// ---- DUTs/ST_DivertConfig.TcDUT
TYPE ST_DivertConfig :
STRUCT
	IntervalToDivert							: UDINT := 1;
	MaxAllowedDivertCount						: UDINT := 4;
	CurrentFunctionCoeffA						: LREAL := 0.5;
	CurrentFunctionCoeffB						: LREAL := 0.17;
	CurrentFunctionCoeffC						: LREAL := 3;
END_STRUCT
END_TYPE;

// ---- DUTs/ST_ExpMoverStatus.TcDUT
TYPE ST_ExpMoverStatus :
STRUCT
	XtsBaseRefData						: REFERENCE TO Tc3_XTS_Utility.ST_PositionInfo;
	HasInterference						: BOOL;
	TrackSectorBndryHeadF			: LREAL;
	TrackSectorBndryTailF			: LREAL;
	TrackSectorCenterHead			: LREAL;
	TrackSectorCenterTail			: LREAL;
	TrackSectorBndryHeadR			: LREAL;
	TrackSectorBndryTailR			: LREAL;
	PartSectorBndryHeadF			: LREAL;
	PartSectorBndryTailF			: LREAL;
	PartSectorCenterHead			: LREAL;
	PartSectorCenterTail			: LREAL;
	PartSectorBndryHeadR			: LREAL;
	PartSectorBndryTailR			: LREAL;
	XtsAdjustedData						: Tc3_XTS_Utility.ST_PositionInfo;
END_STRUCT
END_TYPE

// ---- DUTs/ST_PlcSystem.TcDUT
TYPE ST_PlcSystem :
STRUCT
	nTaskIdx						: DINT;
	nCycleTime					: UDINT;
	TempSysTime					: ULINT;
	SysTime							: ULINT;
	CfgIntervalExec			: UDINT := 2; //x 1 ms task time
END_STRUCT
END_TYPE

// ---- DUTs/ST_SectorsConfig.TcDUT
TYPE ST_SectorsConfig :
STRUCT
	AllSectorsConfig : REFERENCE TO ARRAY[GC.MIN_SECTOR_CT..GC.MAX_SECTOR_CT] OF ST_SectorConfig;
END_STRUCT
END_TYPE

// ---- DUTs/ST_SectorsStatus.TcDUT
TYPE ST_SectorsStatus :
STRUCT
	AllSectorsStatus : REFERENCE TO ARRAY[GC.MIN_SECTOR_CT..GC.MAX_SECTOR_CT] OF ST_SectorStatus;
END_STRUCT
END_TYPE

// ---- DUTs/ST_SwitchStatus.TcDUT
TYPE ST_SwitchStatus :
STRUCT
 	MagnetValue		        AT%Q* 	: INT;
	MagnetEnabled     	        	: BOOL;
    CurrentOutputActual             : LREAL;
    CurrentTheoreticalEstimation    : LREAL;
    CurrentOutputMax                : LREAL;
    PosnCurrentCoeff                : LREAL;
	ShuttleCountAtDivertTrig		: UDINT;
	ShuttleQueueCount				: UDINT;
	ShuttleCountOnShortcut			: UDINT;
END_STRUCT
END_TYPE

// ---- DUTs/ST_SectorConfig.TcDUT
TYPE ST_SectorConfig :
STRUCT
	TrackObjectId			: OTCID;
	PartObjectId	    : OTCID;
	PartObjectIdEnt	    : OTCID;
	PartObjectIdExit    : OTCID;	
	PartSectorStartPosn				: LREAL;
	PartSectorEndPosn				: LREAL;
	TrackSectorStartPosn				: LREAL;
	TrackSectorEndPosn				: LREAL;
	SectorSpansBoundary		: BOOL;
END_STRUCT
END_TYPE

// ---- DUTs/ST_SectorStatus.TcDUT
TYPE ST_SectorStatus :
STRUCT
	MoverIsOnSector			: BOOL;
	MoverCountOnSector		: UDINT;
	MoverEnteredSector		: Tc2_Standard.R_TRIG;
	MoverExitedSector		: Tc2_Standard.F_TRIG;
	SectorLength				: LREAL;
	MoverDistanceFromEnd	: LREAL;
	PercentOfSectorTraversed	: LREAL;
END_STRUCT
END_TYPE

// ---- DUTs/ST_ShortcutConfig.TcDUT
TYPE ST_ShortcutConfig :
STRUCT
	StopAtPowerMat  						: BOOL;
END_STRUCT
END_TYPE

// ---- DUTs/ST_SwitchConfig.TcDUT
TYPE ST_SwitchConfig :
STRUCT
	MagnetOnStartPosition				    : LREAL := 9860; // mm // a little early; 
	MagnetOnEndPosition				    	: LREAL := 10695; // Length of Main Track // mm
	OnInnerLoopOffMagnetPosn				: LREAL	:= 170; //mm
	SwitchCurrentNominal						: LREAL := 5.8; // A (See function for computation)
	CurrentMultFactor							: LREAL := 1310; // Scaling factor for 10V output=25.0A
    UseNominalCurrentVeloSetpoints              : BOOL;
    UseNominalPositionCoeff			            : BOOL := TRUE;
//	PosnCoilResponseTimeCoeffNominal			: LREAL := 0.986;
 	SwitchModeHMI        						: ST_DivertConfig;
 	SwitchModeInternal    						: ST_DivertConfig;
END_STRUCT
END_TYPE;

// ---- DUTs/ST_TrackConfig.TcDUT
TYPE ST_TrackConfig :
STRUCT
	TargetPosnBeforeTrackEnd					: LREAL := 100;
	StopPosPowermat										: LREAL := 7611; // Track Ref; Part Ref ~ 3750 (mm)
	MergeWaitFinishDistance 					: LREAL := 1570;
	MergeWaitAccelDistance						: LREAL; // distance to achieve v_max on the shortcut HD motor region
	ShortcutHDRegionDistance					: LREAL := 2000;
	ShortcutShuttleFullyInPosn 				: LREAL := 1500; // Part Reference (not Track)
	ExpMoverLength										: LREAL := 1200; // roughly 2X SHUTTLE_LENGTH
	MaxLagDistance										: LREAL := 100;
	MergeCollisionRegionDeltaFromL		: LREAL := 2800; // 1715
	MergeCollisionAdvance							: LREAL := 200;
END_STRUCT
END_TYPE

// ---- DUTs/ST_MoverConfig.TcDUT
TYPE ST_MoverConfig EXTENDS ST_MoveOnTrackOptions:
STRUCT
//Velocity (mm/s)
	MaxVelo			: LREAL := 4000;
	NormalVelo		: LREAL := 2700;
	StoppingVelo	: LREAL := 400;
//Acceleration (mm/s^2)
	NormalAccel		: LREAL := MaxVelo;
	MaxAccel		: LREAL := 3*NormalAccel;
//Deceleration (mm/s^2)
	NormalDecel		: LREAL := MaxVelo;	
	MaxDecel		: LREAL := 3*NormalDecel;
//Jerk (mm/s^3)
	NormalJerk		: LREAL := MaxAccel;
	HighJerk			: LREAL := 2*NormalJerk;
	MergeJerk 		: LREAL := 400000;
//Platooning Vars
	VeloComp		: LREAL := 200;
	NormalMoverGap	: LREAL := 750;
	TightMoverGap	: LREAL := 20;
END_STRUCT
END_TYPE

// ---- GVLs/GC.TcGVL
{attribute 'qualified_only'}
VAR_GLOBAL CONSTANT
//Movers-PLC
	nNumMinMovers					: UDINT :=1;
	nNumMaxMovers 					: UDINT :=4; //See General (Persistent, non-constant)

//Movers-MC
	nNumMinMCAxes					: UDINT	:=1;
	nNumMaxMCAxes					: UDINT	:=20;

//Tracks
	nNumMinTracks 					: UDINT :=1; // Do not change - per NC
	OuterFinishPart					: UDINT := 1;
	InnerFinishPart					: UDINT := 2;
	OuterStartPart					: UDINT := 3;	
	nNumMaxTracks 					: UDINT :=3; // Do not change - per NC
	
//Sectors
	MIN_SECTOR_CT										: USINT	:= 1;
	//Make MIN same as first entry
	DIVERTQ_SECTOR_OPART						: USINT := 1;
	DIVERT_DECISION_OPART						: USINT := 2;
	MAG_ON_SECTOR_OPART							: USINT	:= 3; 
	SHORTCUT_ENTRY_SECTOR_IPART 		: USINT := 4; 
	SHORTCUT_ENTRY_HALF_IPART				: USINT := 5; 
	SHORTCUT_CALC_SECTOR_IPART 			: USINT := 6; 
	LOAD_STOP_SECTOR_IPART					: USINT := 7; 
	SHORTCUT_HD_SECTION							: USINT := 8; 
	SHORTCUT_COMPLETE								: USINT := 9; 
	SHORTCUT_EXIT_HALF_IPART				: USINT := 10;
	SHORTCUT_MERGE_COMMAND_WAIT 		: USINT := 11;
	SHORTCUT_MERGE_COMMAND_FLYING 	: USINT := 12;
	SHORTCUT_MERGE_CALC_EXACT 			: USINT := 13;
	INNER_MERGE_TO_FINISH 					: USINT := 14;
	OUTER_SHORTCUT_PROJECTIONFLY		: USINT := 15;
	OUTER_SHORTCUT_PROJECTIONSTAT		: USINT := 16;
	OUTER_PRE_TG_ZONE								: USINT := 17;
	OUTER_TIGHTGAP_ZONE							: USINT := 18;
	OUTER_POST_TG_ZONE							: USINT := 19;
	OUTER_BIGTRACK_END							: USINT := 20;
	OUTER_BIGTRACK_LSMALL						: USINT := 21;
	OUTER_BIGTRACK_MOVE_END					: USINT := 22;
	OUTER_MERGE_COLLISION						: USINT := 23;
	//Make MAX same as last entry
	MAX_SECTOR_CT										: USINT	:= 23;
	
	MIN_TRACKSECTORS_REF : USINT := 1;
	TRACK_SECTORS_STD : USINT := 1;
	TRACK_SECTORS_HEAD : USINT := 2;
	TRACK_SECTORS_TAIL : USINT := 3;
	MAX_TRACKSECTORS_REF : USINT := 3;

	
// Global Position Constants
	SHUTTLE_LENGTH						: LREAL := 600; //mm
END_VAR

// ---- GVLs/GVL_General.TcGVL
VAR_GLOBAL // PERSISTENT
	nNumMovers								: UDINT := 4;
	TotalRuntime							: TIME;
END_VAR

VAR_GLOBAL
	GraphPage												: Tc2_System.T_MaxString := 'https://www.desmos.com/calculator';	

	aStopPositions 									: ARRAY [GC.nNumMinMovers..GC.nNumMaxMovers] OF LREAL;// := [2400, 1700, 1000, 300];

//Configuration
	stMoverConfig										: ST_MoverConfig;
	stTrackGlobalConfig							: ST_TrackConfig;
	stPlanarTrackConfig							: ARRAY[GC.nNumMinTracks..GC.nNumMaxTracks] OF ST_PlanarTrackConfig;
	stTrackShortcutConfig						: ST_ShortcutConfig;
	stSwitchConfig									: ST_SwitchConfig;
	
//XTS - Complete Loop
	XtsCompleteTrackOuterOID				: OTCID := 16#1010480;
	XtsCompleteTrackInnerOID				: OTCID := 16#1010490;
//XTS - Parts
	XtsPartOuterStart								: OTCID := 16#01010020;
	XtsPartInnerFinish							: OTCID := 16#01010170;
	XtsPartOuterFinish							: OTCID := 16#010102C0;
//Planar
	PlanarTrackOuterStart						: OTCID := 16#05120030;
	PlanarTrackInnerFinish					: OTCID := 16#05120020;
	PlanarTrackOuterFinish					: OTCID := 16#05120010;

//Divert
	DivertQueue											: FB_DivertQueue; // Buffer for Divert Requests
	HistoryDivertQueue							: FB_DivertQueue; // Log of all that went through the trigger point
	TempItvlMoverIndex							: UDINT;
	MoverIndexDivertTrig							: UDINT := GC.nNumMinMovers;
	stDivertingMover								: RingBuffer.ST_MoverDivert;
	stMoverDivertInit 							: RingBuffer.ST_MoverDivert; // DO NOT write to this var
	SwitchMagnet										: FB_SwitchMagnet;
	nExitAMoverIsUsingMagnet				: UDINT;
	MagnetControlledByOtherMover		: BOOL;
	ftMagnetControlledByOtherMover	: Tc2_Standard.F_TRIG;
	stSwitchStatus        		    	: ST_SwitchStatus;

//Merge
	MergeQueue											: RingBuffer.RingBufferMoverMerge; // Buffer for Merge events

END_VAR

// ---- GVLs/GVL_Mc3.TcGVL
VAR_GLOBAL	
	TrackSectors					: ARRAY[GC.nNumMinMovers..GC.nNumMaxMovers] OF FB_TrackSectors;
	HeadTrackSectors			: ARRAY[GC.nNumMinMovers..GC.nNumMaxMovers] OF FB_TrackSectors;
	TailTrackSectors			: ARRAY[GC.nNumMinMovers..GC.nNumMaxMovers] OF FB_TrackSectors;
	AllTrackSectors				: FB_AllTrackSectors;

{warning <'bundle FB_Track'>}
	MC_Tracks    		   	 	: ARRAY[GC.nNumMinTracks..GC.nNumMaxTracks] OF Tc3_Mc3PlanarMotion.MC_PlanarTrack;
	MC_Trackfeedback	 		: ARRAY[GC.nNumMinTracks..GC.nNumMaxTracks] OF Tc3_Mc3PlanarMotion.MC_PlanarFeedback;
	TrackTrail 			   		: Tc3_Mc3PlanarMotion.MC_PlanarTrackTrail;
	
{warning <'bundle FB_PlanarMover'>}
	fbPlanarXtsMover			: ARRAY[GC.nNumMinMovers..GC.nNumMaxMovers] OF FB_PlanarXtsMover;
	iMover								: ARRAY[GC.nNumMinMovers..GC.nNumMaxMovers] OF RingBuffer.I_MoverBase;
	aiXpuXtsMover       	: ARRAY[GC.nNumMinMovers..GC.nNumMaxMovers] OF Tc3_XTS_Utility.I_TcIoXtsXpuMover;

	HeadExpMover					: ARRAY[GC.nNumMinMovers..GC.nNumMaxMovers] OF FB_ExpandedMover;
	TailExpMover					: ARRAY[GC.nNumMinMovers..GC.nNumMaxMovers] OF FB_ExpandedMover;
	AllExpMovers					: FB_AllExpMovers;
END_VAR

// ---- ITFs/I_Mover.TcIO
INTERFACE I_Mover (*EXTENDS RingBuffer.I_MoverBase*)

METHOD CycleUpdate : BOOL
VAR_INPUT
END_VAR
END_METHOD

METHOD Init : BOOL
VAR_INPUT
	XtsMover:  I_XtsXlMover1;
	XtsProcessingUnit :  I_XtsProcessingUnit1;
END_VAR
END_METHOD

METHOD JoinNearestTrack : BOOL


VAR

END_VAR
END_METHOD

METHOD LeaveSystemAt : BOOL
VAR_INPUT
	ConnectionOut: REFERENCE TO MC_PlanarTrackConnectionOut;	
END_VAR
END_METHOD

METHOD MoveOnTrack : BOOL
VAR_INPUT
	track: REFERENCE TO MC_PlanarTrack;	
	targetPos: LREAL;
	gap : LREAL; 
	velo : LREAL; 
END_VAR
END_METHOD

PROPERTY MoverOTCID : OTCID
GET
END_GET
SET
END_SET
END_PROPERTY

PROPERTY MoverStopped : BOOL
GET
END_GET
SET
END_SET
END_PROPERTY

PROPERTY P_Dynamics : REFERENCE TO DynamicConstraint_PathXY;
GET
END_GET
END_PROPERTY

PROPERTY P_InSync : Bool
GET
END_GET
END_PROPERTY

PROPERTY P_PlanarFeedback : REFERENCE TO MC_PlanarFeedback
GET
END_GET
END_PROPERTY

PROPERTY P_PlanarMover :   REFERENCE TO  MC_PlanarMover
GET
END_GET
END_PROPERTY

PROPERTY P_TargetTrack : UDINT
GET
END_GET
SET
END_SET
END_PROPERTY

PROPERTY P_TrackSectors : REFERENCE TO FB_TrackSectors
GET
END_GET
SET
END_SET
END_PROPERTY

PROPERTY Rework : BOOL
GET
END_GET
SET
END_SET
END_PROPERTY

METHOD SyncToOtherMover : Bool
VAR_INPUT
	masterSyncPos : LREAL; // Position on the master track
	followerSyncPos : LREAL; // position on the follower track
	PlanarMoverToFollow: REFERENCE TO Tc3_Mc3PlanarMotion.MC_PlanarMover;
	masterTrack : REFERENCE TO Tc3_Mc3PlanarMotion.MC_PlanarTrack; 
	followerTrack : REFERENCE TO Tc3_Mc3PlanarMotion.MC_PlanarTrack; 
	velo : LREAL; 
END_VAR
END_METHOD

METHOD  UpdateXtsTrack
VAR_INPUT
END_VAR
VAR

END_VAR
END_METHOD

PROPERTY XlProcessingUnit : I_XtsProcessingUnit1
GET
END_GET
END_PROPERTY

PROPERTY XtsComFeed : REFERENCE TO  XtsCommandFeedback
GET
END_GET
END_PROPERTY

PROPERTY XtsXlMover :  I_XtsXlMover1
GET
END_GET
END_PROPERTY

END_INTERFACE

// ---- ITFs/I_MoverSector.TcIO
INTERFACE I_MoverSector EXTENDS __SYSTEM.IQueryInterface

PROPERTY P_SectorsConfig : REFERENCE TO ST_SectorsConfig
GET
END_GET
END_PROPERTY

PROPERTY P_SectorsStatus : REFERENCE TO ST_SectorsStatus
GET
END_GET
END_PROPERTY

END_INTERFACE

// ---- POUs/MAIN.TcPOU
PROGRAM MAIN
VAR
	ManMergeCmd				: BOOL;
	bAllDone					: BOOL;
	bStopSequence				: BOOL;
	                    		
	nCase 						: INT;
	nMoveState				  	: ARRAY[GC.nNumMinMovers..GC.nNumMaxMovers] OF INT;
	                    		
	fbXtsEnvironment			: Tc3_XTS_Utility.FB_TcIoXtsEnvironment;
	                    		
	nForCounter					: UDINT;
	M,N,T,Tr					: UDINT;
	dynamics				    : INT;

//Status
	xSimulation					: BOOL := TRUE;
	SystemEnabled				: BOOL;
	stPlcSystem					: ST_PlcSystem;

	IsMoverInBlockingArea		: BOOL;
	nActStopPos					: UINT := 1;
	Fp_error 					: Tc2_Standard.R_TRIG;
	FaultReset					: Tc2_Standard.R_TRIG;
	MoverStop 	AT%I* 			: BOOL;
  ResetSafetyLight AT%Q*      : BOOL;
	MoverStopDone AT%Q*			: BOOL;
	Info 		AT%Q*			: BOOL;
	Operating	AT%Q*			: BOOL;
	Process		AT%Q*			: BOOL;
	Fault		AT%Q*			: BOOL;
	Emergency	AT%Q*			: BOOL;
	                        	
	Voltage1	AT%I*			: UDINT;
	Voltage2	AT%I*			: UDINT;
	                        	
	TcRestart 					: Tc2_Utilities.TC_Restart;
	Restart 					: BOOL;
	busy 						: BOOL;
	fp_start 					: Tc2_Standard.R_TRIG;
	bStartSequence				: BOOL;
	                        	
	Horntimer 					: Tc2_Standard.TP; 
	R_trigHorn 					: Tc2_Standard.R_TRIG;

	StopTime 					: TIME := T#1S;
	StopTimer 					: ARRAY[GC.nNumMinMovers..GC.nNumMaxMovers] OF Tc2_Standard.TON;
	StartTimer 					: ARRAY[GC.nNumMinMovers..GC.nNumMaxMovers] OF BOOL;

	ArcLength 					: ARRAY[GC.nNumMinMovers..GC.nNumMaxMovers] OF LREAL;
	TrackPos					: ARRAY[GC.nNumMinMovers..GC.nNumMaxMovers] OF ARRAY[GC.nNumMinTracks..GC.nNumMaxTracks] OF Tc3_Physics.PositionXYC;
END_VAR

fbXtsEnvironment.Init(bExecute := TRUE);
//Cyclic
M_WritePlanarTrackConfig();
M_UpdateConfigurations();
IF xSimulation THEN
	SystemEnabled	:= TRUE;
ELSE
	SystemEnabled	:= (MoverStop (* SafetyOK *) AND NOT Fault);
END_IF

stPlcSystem.nTaskIdx := GETCURTASKINDEXEX();
IF stPlcSystem.nTaskIdx > 0 THEN
	stPlcSystem.nCycleTime := _TaskInfo[stPlcSystem.nTaskIdx].CycleTime;
	stPlcSystem.SysTime 	:= Tc2_System.F_GetSystemTime();
END_IF

//Command Diverting to Magnet for any designated mover
DivertQueue();
HistoryDivertQueue(); // no removal
MergeQueue();

//Check if any Mover using Magnet;
FOR nExitAMoverIsUsingMagnet :=  GC.nNumMinMovers TO GVL_General.nNumMovers DO
	IF fbPlanarXtsMover[nExitAMoverIsUsingMagnet].P_IsUsingMagnet THEN
		MagnetControlledByOtherMover		:= TRUE;
		EXIT;
	ELSE
		MagnetControlledByOtherMover		:= FALSE;
	END_IF
END_FOR

SwitchMagnet(SafetyPermIntlk := SystemEnabled,
			stSwitchConfig := GVL_General.stSwitchConfig);
ftMagnetControlledByOtherMover(CLK := MagnetControlledByOtherMover);

Emergency :=  MoverStop;
ResetSafetyLight    := NOT MoverStop;

Operating := NOT  MoverStop;
R_trigHorn(clk := Voltage1> 10000 OR Voltage2 >10000);
Horntimer(in:= ( R_trigHorn.Q ) , PT:= T#2S,Q=> info);

IF nCase > 90 THEN
	Process := TRUE;
ELSE 
	Process := FALSE;	
END_IF

IF NOT fbXtsEnvironment.P_IsInitialized THEN
	RETURN;
END_IF

IF NOT MoverStop AND NOT MoverStopDone THEN
	FOR nForCounter:=1 TO nNumMovers DO
		fbPlanarXtsMover[nForCounter].P_Dynamics.SetValuesVADJ(V := stMoverConfig.MaxVelo, A := stMoverConfig.MaxAccel, D := stMoverConfig.MaxDecel, J := stMoverConfig.HighJerk);
		nCase := 140;
		//fbPlanarMover[nForCounter].McPlanarMover.Halt(fbPlanarXtsMover[nForCounter].P_MoverFeedback, fbPlanarXtsMover[nForCounter].P_Dynamics);
	END_FOR		
	MoverStopDone := TRUE;
ELSIF MoverStop THEN
	MoverStopDone := FALSE;
END_IF


TcRestart(
NETID:= '', 
RESTART:= Restart, 
TMOUT:=T#5S , 
BUSY=>busy , 
ERR=> , 
ERRID=> );


fp_start(CLK := bStartSequence);
IF fp_start.Q THEN
	nCase := 10;
	bStartSequence := FALSE;
END_IF

//IsMoverCommandedInShortcut := FALSE;
IsMoverInBlockingArea := FALSE;

bAllDone:= TRUE;
FOR M := GC.nNumMinMovers TO GVL_General.nNumMovers DO///Movers
	StopTimer[M](in:=StartTimer[m],PT:=StopTime);
	GVL_Mc3.fbPlanarXtsMover[M].P_MoverId := M;
	GVL_Mc3.fbPlanarXtsMover[M].P_MoverSort.MoverNumber	:= GVL_Mc3.fbPlanarXtsMover[M].nMoverId;
  GVL_Mc3.aiXpuXtsMover[M]  := fbXtsEnvironment.XpuTcIo(1).MoverTcIo(TO_UINT(M));
  fbPlanarXtsMover[M].iTcIoXtsXpuMover REF= GVL_Mc3.aiXpuXtsMover[M];
	fbPlanarXtsMover[M].Update();
	
	//MoverPos[M].SetValuesXYC(fbPlanarMover[M].McPlanarMover.MCTOPLC.SET.SetPos.x, fbPlanarMover[M].McPlanarMover.MCTOPLC.SET.SetPos.y,fbPlanarMover[M].McPlanarMover.MCTOPLC.SET.SetPos.c);
	
	TR := Tr+1;
	IF Tr = 4 THEN
		Tr :=1;
	END_IF
	{warning <'MoverPhysics does not work'>}
	ArcLength[M] :=GVL_Mc3.MC_Tracks[Tr].GetArcLengthClosestTo(GVL_Mc3.fbPlanarXtsMover[M].P_Physics);
	GVL_Mc3.MC_Tracks[Tr].GetPositionAt(ArcLength[M],TrackPos[M][Tr]);
	
//	IF ABS(GVL_Mc3.fbPlanarXtsMover[M].MoverPhysics.x - TrackPos[M][Tr].x) < 1 AND  ABS(fbPlanarXtsMover[M].MoverPhysics.y - TrackPos[M][Tr].y) < 1 THEN
// 		GVL_Mc3.fbPlanarXtsMover[M].P_XPlanarMover.MoverTrackNr := Tr;
//	END_IF	
	
//	IsMoverCommandedInShortcut := IsMoverCommandedInShortcut OR fbPlanarXtsMover[M].IsCommandedInShortcut;
//	IsMoverInBlockingArea := IsMoverInBlockingArea OR (GVL_Mc3.fbPlanarXtsMover[M].P_PlanarMover.TrackID = GVL_Mc3.MC_Tracks[E_TrackNum.main].MCTOPLC_STD.TrackOID AND 
//														IsBetween(value := GVL_Mc3.fbPlanarXtsMover[M].P_PlanarMover.MoverPos, 
//														minV := GVL_General.stSwitchConfig.fMagnetEntryPosn - GVL_General.stSwitchConfig.MagnetPosnComp, 
//														maxV :=  GVL_General.stSwitchConfig.fMagnetExitPosn + stSwitchConfig.MagnetPosnComp));
	fbPlanarXtsMover[M].P_MoverFeedback.Update();

	Fp_error(CLK := fbPlanarXtsMover[M].P_MC_PlanarMover.Error AND nCase = 100);
	IF Fp_error.Q THEN
		nCase := 140;
		Fault := TRUE;
//		bCmdMagnetOn := FALSE;
	END_IF
END_FOR

FOR T := GC.nNumMinTracks TO GC.nNumMaxTracks DO 
	MC_Tracks[T].Update();
	MC_Trackfeedback[T].Update();
END_FOR

CASE nCase OF
	10:
		Fault := FALSE;
		FOR nForCounter := 1 TO fbXtsEnvironment.XpuTcIo(1).GetPartCount() DO
			fbXtsEnvironment.XpuTcIo(1).PartTcIo(TO_UINT(nForCounter)).TriggerReset();
		END_FOR
		
		nCase := 20;

	20:
		FOR T := GC.nNumMinTracks TO GC.nNumMaxTracks DO 
			MC_Tracks[T].Enable(MC_Trackfeedback[T]);
		END_FOR
				nCase := 30;
		
		
	30: 
		IF MC_Trackfeedback[E_TrackNum.Big].Done AND MC_Trackfeedback[E_TrackNum.Main].Done AND MC_Trackfeedback[E_TrackNum.Small].Done THEN
			nCase := 35;
		END_IF
		
		
	35:
		FOR nForCounter:=GC.nNumMinMovers TO GVL_General.nNumMovers DO
			fbPlanarXtsMover[nForCounter].P_MC_PlanarMover.Reset(fbPlanarXtsMover[nForCounter].P_MoverFeedback);
		END_FOR
		nCase := 36;	
		
		
	36:	
		bAllDone:=TRUE;
		FOR nForCounter:=GC.nNumMinMovers TO GVL_General.nNumMovers DO
			bAllDone:=bAllDone AND fbPlanarXtsMover[nForCounter].P_MoverFeedback.Done;
		END_FOR
		
		IF bAllDone THEN
			nCase := 40;
		END_IF
		
		
	40:
		FOR nForCounter:=GC.nNumMinMovers TO GVL_General.nNumMovers DO
			fbPlanarXtsMover[nForCounter].P_MC_PlanarMover.Enable(fbPlanarXtsMover[nForCounter].P_MoverFeedback);
		END_FOR
		nCase := 50;
	
		
	50:
		bAllDone:=TRUE;
		FOR nForCounter:=GC.nNumMinMovers TO GVL_General.nNumMovers DO
			bAllDone:=bAllDone AND fbPlanarXtsMover[nForCounter].P_MoverFeedback.Done;
		END_FOR
		
		IF bAllDone THEN
			nCase := 60;
		END_IF

	//55:

	60:
		FOR nForCounter:=GC.nNumMinMovers TO GVL_General.nNumMovers DO
			IF nForCounter <= 9 THEN
				fbPlanarXtsMover[nForCounter].JoinTrack(fbPlanarXtsMover[nForCounter].P_MoverFeedback, GVL_Mc3.MC_Tracks[E_TrackNum.Big]);//   Mover[nForCounter].MoverTrackNr]);
			ELSE
				fbPlanarXtsMover[nForCounter].JoinTrack(fbPlanarXtsMover[nForCounter].P_MoverFeedback, GVL_Mc3.MC_Tracks[E_TrackNum.Main]);
			END_IF	
		END_FOR
		
		nCase := 70;
		
	70:
		bAllDone:=TRUE;
		FOR nForCounter:=GC.nNumMinMovers TO GVL_General.nNumMovers DO
			bAllDone:=bAllDone AND fbPlanarXtsMover[nForCounter].P_MoverFeedback.Done;
		END_FOR
		
		IF bAllDone THEN
			nCase := 80;
		END_IF
		
	80:	
		FOR nForCounter:=GC.nNumMinMovers TO GVL_General.nNumMovers DO
			nMoveState[nForCounter] := 0;
			fbPlanarXtsMover[nForCounter].P_MoverOptions.BaseMoveOptions.direction := MC_Direction.mcDirectionPositive;
			fbPlanarXtsMover[nForCounter].P_MoverOptions.BaseMoveOptions.gapMode := MC_GAP_MODE_ON_TRACK.Fast1D;
		END_FOR
		
		nCase := 100;

	100:

		FOR nForCounter:= GC.nNumMinMovers TO GVL_General.nNumMovers DO
			
		//increased accel on shortcut
			IF TrackSectors[nForCounter].SectorStatus[GC.SHORTCUT_HD_SECTION].MoverIsOnSector THEN
				//Increase dynamics on Inner Shortcut
				fbPlanarXtsMover[nForCounter].P_Dynamics.SetValuesVADJ(V := stMoverConfig.NormalVelo, A := stMoverConfig.MaxAccel, D := stMoverConfig.MaxDecel, J := stMoverConfig.HighJerk);
			ELSE
				fbPlanarXtsMover[nForCounter].P_Dynamics.SetValuesVADJ(V := stMoverConfig.NormalVelo, A := stMoverConfig.NormalAccel, D := stMoverConfig.NormalDecel, J := stMoverConfig.NormalJerk);
			END_IF
			

			//Gap Control
			fbPlanarXtsMover[nForCounter].M_EvaluateGap(MoverIndex := nForCounter);

			//Adjust the first mover parameters to induce a platoon
			fbPlanarXtsMover[GC.nNumMinMovers].P_Dynamics.SetValuesVADJ(V := stMoverConfig.NormalVelo-stMoverConfig.VeloComp, A := stMoverConfig.NormalAccel, D := stMoverConfig.NormalDecel, J := stMoverConfig.NormalJerk);

			// allow updating the config per the HMI, when it will not jeopardize the system
			IF NOT TrackSectors[nForCounter].SectorStatus[GC.DIVERT_DECISION_OPART].MoverIsOnSector AND NOT 
				TrackSectors[nForCounter].SectorStatus[GC.SHORTCUT_ENTRY_HALF_IPART].MoverIsOnSector THEN
				stSwitchConfig.SwitchModeInternal		:= 						stSwitchConfig.SwitchModeHMI;
			END_IF
		
			TrackSectors[nForCounter](MoverIndex := nForCounter, MoverRef := iMover[nForCounter]);
//			HeadTrackSectors[nForCounter](MoverIndex := nForCounter, MoverRef := HeadExpMover[nForCounter]);
//			TailTrackSectors[nForCounter](MoverIndex := nForCounter, MoverRef := TailExpMover[nForCounter]);			
			AllTrackSectors(TrackSectorsRef := GVL_Mc3.TrackSectors, HeadTrackSectorsRef := HeadTrackSectors, TailTrackSectorsRef := TailTrackSectors);
			
			HeadExpMover[nForCounter](MoverRef := fbPlanarXtsMover[nForCounter]);
			TailExpMover[nForCounter](MoverRef := fbPlanarXtsMover[nForCounter]);
			AllExpMovers(HeadMoversRef := HeadExpMover, TailMoversRef := TailExpMover);
			
			iMover[nForCounter]	:= fbPlanarXtsMover[nForCounter];
			fbPlanarXtsMover[nForCounter]();
			
			CASE nMoveState[nForCounter] OF
				
				0: // Start-up/Init
					IF fbPlanarXtsMover[nForCounter].P_MoverSort.TrackID = GVL_General.PlanarTrackOuterFinish THEN
						fbPlanarXtsMover[nForCounter].P_MC_PlanarMover.MoveOnTrack(commandFeedback := fbPlanarXtsMover[nForCounter].P_MoverFeedback,
																			targetTrack := GVL_Mc3.MC_Tracks[E_TrackNum.Big],
																			targetPositionOnTrack := GVL_Mc3.MC_Tracks[E_TrackNum.Big].GetLength()-stTrackGlobalConfig.TargetPosnBeforeTrackEnd,
																			constraint := fbPlanarXtsMover[nForCounter].P_Dynamics,
																			options := fbPlanarXtsMover[nForCounter].P_MoverOptions.BaseMoveOptions);
						 nMoveState[nForCounter] 	:= 20;
					ELSIF (fbPlanarXtsMover[nForCounter].P_MoverSort.TrackID = GVL_General.PlanarTrackOuterStart) AND 
								fbPlanarXtsMover[nForCounter].P_XtsPositionInfo.fPartPosition < TrackSectors[nForCounter].P_SectorsConfig[GC.DIVERTQ_SECTOR_OPART].PartSectorStartPosn THEN
						fbPlanarXtsMover[nForCounter].P_MC_PlanarMover.MoveOnTrack(commandFeedback := fbPlanarXtsMover[nForCounter].P_MoverFeedback,
																			targetTrack := GVL_Mc3.MC_Tracks[E_TrackNum.Main],
																			targetPositionOnTrack := GVL_Mc3.MC_Tracks[E_TrackNum.Main].GetLength()-stTrackGlobalConfig.TargetPosnBeforeTrackEnd,
																			constraint := fbPlanarXtsMover[nForCounter].P_Dynamics,
																			options := fbPlanarXtsMover[nForCounter].P_MoverOptions.BaseMoveOptions);
						 nMoveState[nForCounter] 	:= 10;
					END_IF
					
				5: // In Recirc - from Big to Main Track - departing Gap Transition Zone - this Move command could be cyclic
					IF stPlcSystem.TempSysTime = 0 XOR stPlcSystem.TempSysTime = stPlcSystem.SysTime THEN
						stPlcSystem.TempSysTime := stPlcSystem.SysTime + (stPlcSystem.CfgIntervalExec * stPlcSystem.nCycleTime); //next valid clock to issue move command again
						fbPlanarXtsMover[nForCounter].P_eMerge		:= E_MergeType.NoMerge;
						fbPlanarXtsMover[nForCounter].P_MasterSyncId	:= 0;
						fbPlanarXtsMover[nForCounter].P_MasterSyncPosition	:= 0;
						fbPlanarXtsMover[nForCounter].P_MC_PlanarMover.MoveOnTrack(commandFeedback := fbPlanarXtsMover[nForCounter].P_MoverFeedback,
																		targetTrack := GVL_Mc3.MC_Tracks[E_TrackNum.Main],
																		targetPositionOnTrack := GVL_Mc3.MC_Tracks[E_TrackNum.Main].GetLength()-stTrackGlobalConfig.TargetPosnBeforeTrackEnd,
																		constraint := fbPlanarXtsMover[nForCounter].P_Dynamics, 
																		options := fbPlanarXtsMover[nForCounter].P_MoverOptions.BaseMoveOptions);
					END_IF
																		
					//Continuously call the above move command while GapInTransition TRUE (otherwise it's a one-shot command)
					IF NOT fbPlanarXtsMover[nForCounter].P_MoverOptions.GapInTransition THEN
						stPlcSystem.TempSysTime		:= 0;
						nMoveState[nForCounter] 	:= 10;
					END_IF

				10: //Trig state for decision to divert
					IF TrackSectors[nForCounter].afbSector[GC.DIVERTQ_SECTOR_OPART].stSectorStatus.MoverEnteredSector.Q THEN
						GVL_General.stSwitchStatus.ShuttleCountAtDivertTrig		:= GVL_General.stSwitchStatus.ShuttleCountAtDivertTrig +1; //always MODing this; don't need to decrement
						TempItvlMoverIndex	:= ((GVL_General.stSwitchStatus.ShuttleCountAtDivertTrig MOD GVL_General.stSwitchConfig.SwitchModeInternal.IntervalToDivert) +1); // capture the index
					//	AllTrackSectors.M_UpdateSectorCounts(SectorNr := GC.SHORTCUT_CALC_SECTOR_IPART);
						MoverIndexDivertTrig			:= fbPlanarXtsMover[nForCounter].P_MoverId; // regardless of the command to divert, log the MoverID
						DivertQueue.M_UpdateAtTrig();
						nMoveState[nForCounter] 	:= 12;
					END_IF
					
				12: // Command to move needs to be given early
					IF TrackSectors[nForCounter].afbSector[GC.DIVERT_DECISION_OPART].stSectorStatus.MoverEnteredSector.Q THEN
						DivertQueue.RemoveObjFromBuffer();
						nMoveState[nForCounter] 	:= 13;
					END_IF
				
				13:				
				IF (DivertQueue.P_LastObjectRemoved.MoverID <> 0) THEN // Valid MoverID must be obtained by Remove op in previous step
					IF SwitchMagnet.P_PermIntlkOK AND NOT MagnetControlledByOtherMover AND fbPlanarXtsMover[nForCounter].P_CmdDivert AND 
						(fbPlanarXtsMover[nForCounter].P_XtsPositionInfo.fPartPosition < GVL_Mc3.TrackSectors[nForCounter].P_SectorsConfig[GC.MAG_ON_SECTOR_OPART].PartSectorStartPosn)
						AND (stDivertingMover.SysTime <> DivertQueue.P_LastObjectRemoved.SysTime) THEN
							// Divert Move command
							stDivertingMover	:= DivertQueue.P_LastObjectRemoved;
							fbPlanarXtsMover[stDivertingMover.MoverID].P_MC_PlanarMover.MoveOnTrack(commandFeedback := fbPlanarXtsMover[stDivertingMover.MoverID].P_MoverFeedback,
																				targetTrack := GVL_Mc3.MC_Tracks[E_TrackNum.Small],
																				targetPositionOnTrack := (GVL_Mc3.MC_Tracks[E_TrackNum.Small].GetLength() - GC.SHUTTLE_LENGTH) / 2, // midpoint of shortcut
																				constraint := fbPlanarXtsMover[stDivertingMover.MoverID].P_Dynamics,
																				options := fbPlanarXtsMover[stDivertingMover.MoverID].P_MoverOptions.BaseMoveOptions);									
							nMoveState[nForCounter] 	:= 30; //Diverting Mover
					ELSIF NOT fbPlanarXtsMover[nForCounter].P_CmdDivert THEN
							nMoveState[nForCounter] 	:= 15;
					END_IF
				END_IF
	
				15: // In Recirc - from Main to Big Track
					fbPlanarXtsMover[nForCounter].P_MC_PlanarMover.MoveOnTrack(commandFeedback := fbPlanarXtsMover[nForCounter].P_MoverFeedback,
																		targetTrack := GVL_Mc3.MC_Tracks[E_TrackNum.Big],
																		targetPositionOnTrack := GVL_Mc3.MC_Tracks[E_TrackNum.Big].GetLength()-stTrackGlobalConfig.TargetPosnBeforeTrackEnd,
																		constraint := fbPlanarXtsMover[nForCounter].P_Dynamics,
																		options := fbPlanarXtsMover[nForCounter].P_MoverOptions.BaseMoveOptions);
					 nMoveState[nForCounter] 	:= 20;				
					
				20:
					IF TrackSectors[nForCounter].afbSector[GC.OUTER_BIGTRACK_END].stSectorStatus.MoverEnteredSector.Q THEN
						nMoveState[nForCounter]     := 5;
					END_IF				

				30: // Match the move command with the shuttle that is commanded to divert
					SwitchMagnet.M_EvaluateInlineCommands();
					
					IF ftMagnetControlledByOtherMover.Q THEN
						nMoveState[nForCounter] 	:= 40;
					END_IF
			
				40: // Route through shortcut
					IF TrackSectors[nForCounter].afbSector[GC.LOAD_STOP_SECTOR_IPART].stSectorStatus.MoverEnteredSector.Q THEN
						IF stTrackShortcutConfig.StopAtPowerMat THEN
							nMoveState[nForCounter] := 90;
						ELSE
							nMoveState[nForCounter] := 50;
						END_IF					
					END_IF
					
				50: //Pre-Merge state
				IF NOT AllTrackSectors.P_AMoverIsOnSector[GC.OUTER_BIGTRACK_LSMALL] 
						(*AND stSwitchConfig.SwitchModeInternal.MaxAllowedDivertCount = GVL_General.nNumMovers*) THEN
					fbPlanarXtsMover[nForCounter].P_eMerge := E_MergeType.FlyingMergeMoveOnTrack;

					fbPlanarXtsMover[nForCounter].P_MC_PlanarMover.MoveOnTrack(commandFeedback := fbPlanarXtsMover[nForCounter].P_MoverFeedback,
																		targetTrack := GVL_Mc3.MC_Tracks[E_TrackNum.Small],
																		targetPositionOnTrack := GVL_Mc3.MC_Tracks[E_TrackNum.Small].GetLength()-stTrackGlobalConfig.TargetPosnBeforeTrackEnd,
																		constraint := fbPlanarXtsMover[nForCounter].P_Dynamics,
																		options := fbPlanarXtsMover[nForCounter].P_MoverOptions.BaseMoveOptions);

					nMoveState[nForCounter] := 75;
					//Sync to Master ExpMover
				ELSIF TrackSectors[nForCounter].afbSector[GC.SHORTCUT_MERGE_COMMAND_FLYING].stSectorStatus.MoverEnteredSector.Q THEN
					//Nonzero means there is valid Master Mover data
					IF MergeQueue.P_LastObjectRemoved.MoverID <> 0 THEN
					fbPlanarXtsMover[nForCounter].P_eMerge				:= E_MergeType.FlyingMergeMoveSyncd;
						fbPlanarXtsMover[nForCounter].P_MasterSyncId := MergeQueue.P_LastObjectRemoved.MoverID;
//						IF MergeQueue.P_LastObjectRemoved.ExpMoverType = E_ExpMover.Head THEN
//							fbPlanarXtsMover[nForCounter].P_MasterSyncPosition	:= HeadExpMover[fbPlanarXtsMover[nForCounter].P_MasterSyncId].stExpMoverStatus.TrackSectorCenterHead;
//						ELSIF MergeQueue.P_LastObjectRemoved.ExpMoverType = E_ExpMover.Tail THEN
//							fbPlanarXtsMover[nForCounter].P_MasterSyncPosition	:= TailExpMover[fbPlanarXtsMover[nForCounter].P_MasterSyncId].stExpMoverStatus.TrackSectorCenterTail;
//						END_IF
							// use raw mover reference; likely need some position compensation, i.e, stTrackGlobalConfig.ExpMoverLength;
							fbPlanarXtsMover[nForCounter].P_MasterSyncPosition	:= fbPlanarXtsMover[fbPlanarXtsMover[nForCounter].P_MasterSyncId].P_XtsPositionInfo.fTrackPosition;							
						MergeQueue.ClearLastRemoved(); // master sync data consumed by slave
						nMoveState[nForCounter] := 72;					
					END_IF
					
				ELSIF TrackSectors[nForCounter].afbSector[GC.SHORTCUT_MERGE_COMMAND_WAIT].stSectorStatus.MoverEnteredSector.Q OR 
					stTrackShortcutConfig.StopAtPowerMat THEN
					fbPlanarXtsMover[nForCounter].P_eMerge := E_MergeType.MergeFromStaticSyncd;
					
					fbPlanarXtsMover[nForCounter].P_MC_PlanarMover.MoveOnTrack(commandFeedback := fbPlanarXtsMover[nForCounter].P_MoverFeedback,
																		targetTrack := GVL_Mc3.MC_Tracks[E_TrackNum.Small],
																		targetPositionOnTrack := GVL_Mc3.MC_Tracks[E_TrackNum.Small].GetLength()-stTrackGlobalConfig.MergeWaitFinishDistance-stTrackGlobalConfig.MergeWaitAccelDistance,
																		constraint := fbPlanarXtsMover[nForCounter].P_Dynamics,
																		options := fbPlanarXtsMover[nForCounter].P_MoverOptions.BaseMoveOptions);

					nMoveState[nForCounter] := 73;
				END_IF

				60: // Merge - Gear In
 //merge with gap zero
					//issue commmand to sync 
//					masterSyncPos := GVL_Mc.MC_Tracks[E_TrackNum.Big].GetLength()-100;
//					masterPosAtSync := Mover[moverInFront].MoverPos; 
//					followSyncPos := GVL_Mc.MC_Tracks[E_TrackNum.Small].GetLength()-1000;
//					followerPosAtSync :=Mover[1].MoverPos; 
//					fbMover[nForCounter].SyncToOtherMover( 
//						masterSyncPos := masterSyncPos,
//						masterTrack := GVL_Mc.MC_Tracks[E_TrackNum.Big],
//						followerSyncPos := followSyncPos,
//						followerTrack := GVL_Mc.MC_Tracks[e_TrackNum.Small],
//						PlanarMoverToFollow := fbMover[moverInFront].P_PlanarMover,
//						velo:= velo);
//						nMoveState[nForCounter] := 80; 
//					aggressiveDynamics.SetValuesVADJ(4000,4000,8000,400000); 
//					fbMover[nForCounter].P_Dynamics := aggressiveDynamics;
					//fbMover[nForCounter].MoveOnTrack(GVL_Mc.MC_Tracks[E_TrackNum.Main],  GVL_Mc.MC_Tracks[E_TrackNum.Main].GetLength()-500,900,velo);				
				
//					IF fbPlanarXtsMover[nForCounter].P_eMerge <> E_MergeType.NoMerge THEN
						fbPlanarXtsMover[nForCounter].P_Dynamics.SetValuesVADJ(V := stMoverConfig.NormalVelo, A := stMoverConfig.MaxAccel, D := stMoverConfig.MaxDecel, J := stMoverConfig.MergeJerk);
						
						fbPlanarXtsMover[nForCounter].P_MC_PlanarMover.GearInPosOnTrackWithMasterMover(
								commandFeedback:= fbPlanarXtsMover[nForCounter].P_PlanarFeedbackGearMM, 
								masterMover:= fbPlanarXtsMover[fbPlanarXtsMover[nForCounter].P_MasterSyncId].P_MC_PlanarMover,
								trackTrail:= fbPlanarXtsMover[nForCounter].P_SyncTrail,
								masterSyncPosition:= fbPlanarXtsMover[nForCounter].P_MasterSyncPosition,
								masterSyncPositionTrack:= GVL_Mc3.MC_Tracks[E_TrackNum.Big], 
								slaveSyncPosition:= fbPlanarXtsMover[nForCounter].P_XtsPositionInfo.fTrackPosition,
								slaveSyncPositionTrack:= GVL_Mc3.MC_Tracks[E_TrackNum.Small], 
								constraint:= fbPlanarXtsMover[nForCounter].P_Dynamics, 
								options:= fbPlanarXtsMover[nForCounter].P_MoverOptions.GearInMasterMoverOptions);
								nMoveState[nForCounter] := 74;
//					END_IF
						//fbPlanarXtsMover[nForCounter].P_InSync THEN				

				61:
				IF fbPlanarXtsMover[nForCounter].P_MoverFeedback.Done AND ManMergeCmd THEN
					ManMergeCmd	:= FALSE;
					nMoveState[nForCounter] := 75; // 62
				END_IF
					
				62:// Permissive to Merge
//					IF NOT AllTrackSectors.P_AMoverIsOnSector[GC.OUTER_MERGE_COLLISION] THEN
//						nMoveState[nForCounter] := 63;
//					END_IF

				63://Merge from Inner to Outer
//						fbPlanarXtsMover[nForCounter].P_MC_PlanarMover.MoveOnTrack(commandFeedback := fbPlanarXtsMover[nForCounter].P_MoverFeedback,
//																			targetTrack := GVL_Mc3.MC_Tracks[E_TrackNum.Small],
//																			targetPositionOnTrack := GVL_Mc3.MC_Tracks[E_TrackNum.Small].GetLength()-stTrackGlobalConfig.TargetPosnBeforeTrackEnd,
//																			constraint := fbPlanarXtsMover[nForCounter].P_Dynamics,
//																			options := fbPlanarXtsMover[nForCounter].P_MoverOptions.BaseMoveOptions);
//						nMoveState[nForCounter] := 75;
				
				75: //Reset Command On Exit
						IF TrackSectors[nForCounter].afbSector[GC.INNER_MERGE_TO_FINISH].stSectorStatus.MoverEnteredSector.Q THEN
							stSwitchStatus.ShuttleQueueCount := stSwitchStatus.ShuttleQueueCount -1;
							nMoveState[nForCounter] := 5;
						END_IF
				
				90: // Stopped at Powermat Station
					IF fbPlanarXtsMover[nForCounter].P_MoverFeedback.Done THEN
						StartTimer[nForCounter] := TRUE;
						nMoveState[nForCounter] := 100;
					END_IF
					
				100:
					IF StopTimer[nForCounter].Q THEN
						StartTimer[nForCounter] := FALSE;
						nMoveState[nForCounter] := 50;
					END_IF
				END_CASE
		
		END_FOR

		IF bStopSequence AND NOT(IsMoverInBlockingArea) THEN
			nCase := 110;
			bStopSequence := FALSE;
		END_IF
		110:
			N:= nNumMovers;
			FOR nForCounter:=1 TO nNumMovers DO		
				GVL_General.aStopPositions[nForCounter] := TO_LREAL(  fbXtsEnvironment.XpuTcIo(1).MoverTcIo(TO_UINT(N)).GetSimulatedStartUpPosition());
				N := N -1;
			END_FOR
			nCase := 120;
		
		120:	
			nActStopPos := UDINT_TO_UINT(GC.nNumMaxMovers-GVL_General.nNumMovers+1);
			FOR nForCounter:=1 TO nNumMovers DO
				fbPlanarXtsMover[nForCounter].P_Dynamics.SetValuesVADJ(V := stMoverConfig.StoppingVelo, A := stMoverConfig.NormalAccel, D := stMoverConfig.NormalDecel, J := stMoverConfig.NormalJerk);
				nMoveState[nForCounter] := 0;
				fbPlanarXtsMover[nForCounter].P_MC_PlanarMover.MoveOnTrack(fbPlanarXtsMover[nForCounter].P_MoverFeedback, GVL_Mc3.MC_Tracks[E_TrackNum.Main], 300, fbPlanarXtsMover[nForCounter].P_Dynamics, fbPlanarXtsMover[nForCounter].P_MoverOptions.BaseMoveOptions);
			END_FOR

			nCase:= 130; 
		130:
			FOR nForCounter:=1 TO GC.nNumMaxMovers - (GVL_General.nNumMovers-GC.nNumMaxMovers)  DO
				CASE nMoveState[nForCounter] OF
					0:								
						
						IF GVL_Mc3.fbPlanarXtsMover[nForCounter].P_MoverSort.MoverPos < 300 AND GVL_Mc3.fbPlanarXtsMover[nForCounter].P_MoverSort.TrackID = GVL_Mc3.MC_Tracks[E_TrackNum.main].MCTOPLC_STD.TrackOID THEN
							fbPlanarXtsMover[nForCounter].P_MoverOptions.BaseMoveOptions.gap:= stMoverConfig.TightMoverGap;
							fbPlanarXtsMover[nForCounter].P_MC_PlanarMover.MoveOnTrack(commandFeedback := fbPlanarXtsMover[nForCounter].P_MoverFeedback,
																				targetTrack := GVL_Mc3.MC_Tracks[E_TrackNum.Main],
																				targetPositionOnTrack := aStopPositions[nActStopPos],
																				constraint := fbPlanarXtsMover[nForCounter].P_Dynamics,
																				options := fbPlanarXtsMover[nForCounter].P_MoverOptions.BaseMoveOptions);									
							nActStopPos := nActStopPos + 1;
							nMoveState[nForCounter] := 10;
						END_IF
				END_CASE
			END_FOR
		
			bAllDone := TRUE;
			FOR nForCounter:=1 TO nNumMovers DO
				IF NOT(fbPlanarXtsMover[nForCounter].P_MoverFeedback.Done OR fbPlanarXtsMover[nForCounter].P_MoverFeedback.Error) THEN
					bAllDone := FALSE;
					EXIT;
				END_IF
			END_FOR
			
			IF bAllDone THEN
				nCase := 150;
			END_IF
		
		140:
			FOR nForCounter:=1 TO nNumMovers DO
				fbPlanarXtsMover[nForCounter].P_MC_PlanarMover.Halt(fbPlanarXtsMover[nForCounter].P_MoverFeedback, fbPlanarXtsMover[nForCounter].P_Dynamics);
			END_FOR	
			
			nCase := 145;
			
		145:
			bAllDone := TRUE;
			FOR nForCounter:=1 TO nNumMovers DO
				IF NOT(fbPlanarXtsMover[nForCounter].P_MoverFeedback.Done OR fbPlanarXtsMover[nForCounter].P_MoverFeedback.Error) THEN
					bAllDone := FALSE;
					EXIT;
				END_IF
			END_FOR
			
			IF bAllDone THEN
				nCase := 150;
			END_IF
		
		//Disable
		150:
			FOR nForCounter:=1 TO nNumMovers DO
				fbPlanarXtsMover[nForCounter].P_MC_PlanarMover.Disable(fbPlanarXtsMover[nForCounter].P_MoverFeedback);
			END_FOR
				
			nCase := 0;
END_CASE

FaultReset(CLK := MoverStop);

IF FaultReset.Q THEN
	Fault	:= FALSE;
END_IF

METHOD M_UpdateConfigurations
stTrackGlobalConfig.MergeWaitAccelDistance := 
F_PosnDisp(Accel := stMoverConfig.MaxAccel, 
								VeloFinal := stMoverConfig.NormalVelo, 
								VeloInit := 0);
END_METHOD

METHOD M_WritePlanarTrackConfig
stPlanarTrackConfig[E_TrackNum.Big].MCTrack				:= GVL_Mc3.MC_Tracks[E_TrackNum.Big].MCTOPLC_STD;
stPlanarTrackConfig[E_TrackNum.Small].MCTrack			:= GVL_Mc3.MC_Tracks[E_TrackNum.Small].MCTOPLC_STD;
stPlanarTrackConfig[E_TrackNum.Main].MCTrack			:= GVL_Mc3.MC_Tracks[E_TrackNum.Main].MCTOPLC_STD;
                                                    	
stPlanarTrackConfig[E_TrackNum.Big].TrackIndex			:= E_TrackNum.Big;
stPlanarTrackConfig[E_TrackNum.Small].TrackIndex		:= E_TrackNum.Small;
stPlanarTrackConfig[E_TrackNum.Main].TrackIndex			:= E_TrackNum.Main;
END_METHOD

END_PROGRAM

// ---- POUs/FUNs/F_PosnDisp.TcPOU
FUNCTION F_PosnDisp : LREAL
VAR_INPUT
	VeloInit 	: LREAL;
	VeloFinal	: LREAL;
	Accel		: LREAL;
END_VAR
VAR
END_VAR

IF Accel <> 0 THEN
	F_PosnDisp := (EXPT(VeloFinal,2) - EXPT(VeloInit,2)) / (2*Accel);
END_IF

END_FUNCTION

// ---- POUs/FBs/FB_DivertQueue.TcPOU
FUNCTION_BLOCK FB_DivertQueue EXTENDS RingBuffer.RingBufferMoverDivert
VAR
//	nForCounterInterval			: UDINT;
	MoverDivert							: RingBuffer.ST_MoverDivert;
END_VAR

METHOD M_UpdateAtTrig
VAR_INST
	stDivertLogMover								: RingBuffer.ST_MoverDivert;
END_VAR
stDivertLogMover.MoverID							:= MoverIndexDivertTrig;
IF (stSwitchStatus.ShuttleQueueCount < GVL_General.stSwitchConfig.SwitchModeInternal.MaxAllowedDivertCount) THEN // permissives to allow a mover to divert
		stDivertLogMover.Divert								:= RingBuffer.E_Divert.Divert;
	IF (TempItvlMoverIndex = GVL_General.stSwitchConfig.SwitchModeInternal.IntervalToDivert) THEN
		stDivertLogMover.DivertOnInterval													:= TRUE;
		stSwitchStatus.ShuttleQueueCount := stSwitchStatus.ShuttleQueueCount + 1;
		fbPlanarXtsMover[stDivertLogMover.MoverID].P_CmdDivert		:= (stDivertLogMover.Divert = RingBuffer.E_Divert.Divert) AND stDivertLogMover.DivertOnInterval;
		HistoryDivertQueue.AddObjToBuffer(RefObject := stDivertLogMover);
	END_IF
END_IF

DivertQueue.AddObjToBuffer(RefObject := stDivertLogMover);
stDivertLogMover					:= stMoverDivertInit;
END_METHOD

PROPERTY P_MoverDivert : REFERENCE TO ST_MoverDivert
GET
P_MoverDivert REF= MoverDivert;
END_GET
END_PROPERTY

END_FUNCTION_BLOCK

// ---- POUs/FBs/FB_SwitchMagnet.TcPOU
FUNCTION_BLOCK FB_SwitchMagnet

VAR_INPUT
	stSwitchConfig				: REFERENCE TO ST_SwitchConfig := GVL_General.stSwitchConfig;
	ShuttleVelocity				: REFERENCE TO LREAL := GVL_General.stMoverConfig.NormalVelo;
	SafetyPermIntlk				: REFERENCE TO BOOL;
END_VAR
//VAR_IN_OUT
//	MoverRef						: 
//END_VAR
VAR
	TimeoutTime					: TIME := T#3S;
	pwm							: FB_PWM;
	Command	 		  			: BOOL;
	Timeout						: TON;
	PermIntlkOK					: BOOL;
END_VAR
VAR_OUTPUT
	MagnetIsOn					: BOOL;
END_VAR

_M_EvaluatePermIntlk();
_M_EvaluateCommands();

//Configuration
IF GVL_General.stSwitchConfig.UseNominalCurrentVeloSetpoints THEN
    GVL_General.stSwitchStatus.CurrentTheoreticalEstimation     := GVL_General.stSwitchConfig.SwitchCurrentNominal;
ELSE
    GVL_General.stSwitchStatus.CurrentTheoreticalEstimation     := F_CurrentVelocity(Velocity := GVL_General.stMoverConfig.NormalVelo, a := GVL_General.stSwitchConfig.SwitchModeHMI.CurrentFunctionCoeffA, b := GVL_General.stSwitchConfig.SwitchModeHMI.CurrentFunctionCoeffB, c := GVL_General.stSwitchConfig.SwitchModeHMI.CurrentFunctionCoeffC);
END_IF

GVL_General.stSwitchStatus.CurrentOutputMax     := GVL_General.stSwitchStatus.CurrentTheoreticalEstimation;

//Output
IF PermIntlkOK AND Command THEN
	GVL_General.stSwitchStatus.MagnetValue := LREAL_TO_INT(GVL_General.stSwitchStatus.CurrentOutputMax*stSwitchConfig.CurrentMultFactor);
ELSE
	GVL_General.stSwitchStatus.MagnetValue := 0;
END_IF

MagnetIsOn	:= (GVL_General.stSwitchStatus.MagnetValue > 0);

IF stSwitchConfig.CurrentMultFactor <> 0 THEN
    GVL_General.stSwitchStatus.CurrentOutputActual  := GVL_General.stSwitchStatus.MagnetValue / stSwitchConfig.CurrentMultFactor;
END_IF

pwm();

//Use Magnet feedback to this timer; set preset time based on mover velocity
Timeout(IN := MagnetIsOn, PT := TimeoutTime);

METHOD PRIVATE _M_EvaluateCommands
VAR_INST
	nForCounter		: UDINT;
END_VAR
IF NOT PermIntlkOK OR Timeout.Q THEN
	Command		:= FALSE;
END_IF
END_METHOD

METHOD PRIVATE _M_EvaluatePermIntlk
PermIntlkOK	:= SafetyPermIntlk AND NOT Timeout.Q;
END_METHOD

METHOD M_EvaluateInlineCommands
IF stDivertingMover.MoverID <> 0 THEN
	IF GVL_Mc3.TrackSectors[stDivertingMover.MoverID].SectorStatus[GC.MAG_ON_SECTOR_OPART].MoverIsOnSector THEN
		Command								:= TRUE;
		fbPlanarXtsMover[stDivertingMover.MoverID].P_IsUsingMagnet := TRUE;
	ELSIF GVL_Mc3.TrackSectors[stDivertingMover.MoverID].SectorStatus[GC.MAG_ON_SECTOR_OPART].MoverExitedSector.Q THEN
		Command								:= FALSE; // Any mover exiting the Magnet drops the command
		fbPlanarXtsMover[stDivertingMover.MoverID].P_CmdDivert			:= FALSE;
		fbPlanarXtsMover[stDivertingMover.MoverID].P_IsUsingMagnet 	:= FALSE;
	END_IF
END_IF
END_METHOD

PROPERTY P_PermIntlkOK : BOOL
GET
P_PermIntlkOK := PermIntlkOK;
END_GET
SET
PermIntlkOK := P_PermIntlkOK;
END_SET
END_PROPERTY

END_FUNCTION_BLOCK

// ---- POUs/FUNs/F_CurrentVelocity.TcPOU
FUNCTION F_CurrentVelocity : LREAL
VAR_INPUT
    Velocity    : LREAL;
	a			: LREAL := 1.1;
	b			: LREAL := 0.1;
	c			: LREAL := 5.8;
END_VAR

F_CurrentVelocity  := a*EXPT((Velocity/1000),2) + b*(Velocity/1000) + c;

END_FUNCTION

// ---- POUs/FBs/FB_TrackSectors.TcPOU
FUNCTION_BLOCK FB_TrackSectors IMPLEMENTS I_MoverSector
// VAR_INPUT
// END_VAR                
VAR                    
//	InitDone						: BOOL;
	SectorIndex						: UDINT;
                       
//Configurations       
	SectorConfig					: ARRAY[GC.MIN_SECTOR_CT..GC.MAX_SECTOR_CT] OF ST_SectorConfig;
	SectorsConfig					: ST_SectorsConfig;
                       
	afbSector								: ARRAY[GC.MIN_SECTOR_CT..GC.MAX_SECTOR_CT] OF FB_TrackSector;
	
	LinkedMoveList 				: ARRAY[GC.MIN_SECTOR_CT..GC.MAX_SECTOR_CT] OF RingBuffer.RingBufferLinkedListEntry;
	iMover								: RingBuffer.ST_IDLinkedListEntry;
END_VAR
VAR_IN_OUT
	MoverIndex						: UDINT;
	MoverRef						: RingBuffer.I_MoverBase; // I_Mover
END_VAR
VAR_OUTPUT
	SectorStatus					: ARRAY[GC.MIN_SECTOR_CT..GC.MAX_SECTOR_CT] OF ST_SectorStatus;
	SectorsStatus					: ST_SectorsStatus;
END_VAR

//IF NOT InitDone THEN
	_M_Configurations();
//END_IF

iMover.iMover := MoverRef;

_M_UpdateStatus();

FOR SectorIndex := GC.MIN_SECTOR_CT TO GC.MAX_SECTOR_CT DO
	//SectorLists
	LinkedMoveList[SectorIndex]();	

	//Planar Mover
	afbSector[SectorIndex].P_MoverSort			:= GVL_Mc3.fbPlanarXtsMover[MoverIndex].P_MoverSort;

	//XTS Mover Reference
	IF MoverRef <> 0 THEN
		afbSector[SectorIndex].P_XtsPositionInfo		:= MoverRef.P_XtsPositionInfo;
	END_IF
	
	//Sector Configuration
	afbSector[SectorIndex].P_TrackSectorConfig	:= SectorConfig[SectorIndex];

	//FB calls
	afbSector[SectorIndex](refPlanarTracks := GVL_General.stPlanarTrackConfig);
END_FOR

METHOD _M_Configurations
IF (GVL_General.XtsCompleteTrackOuterOID <> 0) AND (GVL_General.XtsCompleteTrackInnerOID <> 0) THEN

{warning <'Make this a function of velocity; it's not that sensitive to current'>}
//IF GVL_General.stSwitchConfig.UseNominalPositionCoeff THEN
//	GVL_General.stSwitchStatus.PosnCurrentCoeff                                 := GVL_General.stSwitchConfig.PosnCoilResponseTimeCoeffNominal;
//ELSE (* NOT GVL_General.stSwitchConfig.UseHMINominalSetpoints *)
//	GVL_General.stSwitchStatus.PosnCurrentCoeff                                 := PositionF_CurrentCoeff(Current := GVL_General.stSwitchStatus.CurrentOutputMax);
//END_IF

	SectorConfig[GC.DIVERTQ_SECTOR_OPART].PartObjectId								:= GVL_General.XtsPartOuterStart;
	SectorConfig[GC.DIVERTQ_SECTOR_OPART].PartSectorStartPosn				:= SectorConfig[GC.DIVERT_DECISION_OPART].PartSectorStartPosn - GC.SHUTTLE_LENGTH;
	SectorConfig[GC.DIVERTQ_SECTOR_OPART].PartSectorEndPosn			 		:= SectorConfig[GC.DIVERT_DECISION_OPART].PartSectorStartPosn;
	SectorConfig[GC.DIVERTQ_SECTOR_OPART].TrackSectorStartPosn				:= 0; 
	SectorConfig[GC.DIVERTQ_SECTOR_OPART].TrackSectorEndPosn 				:= 0;

	SectorConfig[GC.DIVERT_DECISION_OPART].PartObjectId						:= GVL_General.XtsPartOuterStart;
	SectorConfig[GC.DIVERT_DECISION_OPART].PartSectorStartPosn			:= F_PosnInitial(VeloInit := GVL_General.stMoverConfig.NormalVelo, VeloFinal := 0, Accel := GVL_General.stMoverConfig.NormalDecel, PosnFinal := SectorConfig[GC.MAG_ON_SECTOR_OPART].PartSectorStartPosn);
	SectorConfig[GC.DIVERT_DECISION_OPART].PartSectorEndPosn			 	:= SectorConfig[GC.MAG_ON_SECTOR_OPART].PartSectorStartPosn;
	SectorConfig[GC.DIVERT_DECISION_OPART].TrackSectorStartPosn			:= 0; 
	SectorConfig[GC.DIVERT_DECISION_OPART].TrackSectorEndPosn 			:= 0;

	SectorConfig[GC.MAG_ON_SECTOR_OPART].PartObjectId						:= GVL_General.XtsPartOuterStart;
	SectorConfig[GC.MAG_ON_SECTOR_OPART].PartSectorStartPosn			:= GVL_General.stSwitchConfig.MagnetOnStartPosition;
	SectorConfig[GC.MAG_ON_SECTOR_OPART].PartSectorEndPosn			 	:= GVL_General.stSwitchConfig.MagnetOnEndPosition;
	SectorConfig[GC.MAG_ON_SECTOR_OPART].TrackSectorStartPosn			:= GVL_General.stSwitchConfig.MagnetOnStartPosition;
	SectorConfig[GC.MAG_ON_SECTOR_OPART].TrackSectorEndPosn 			:= GVL_General.stSwitchConfig.MagnetOnEndPosition;
	SectorConfig[GC.MAG_ON_SECTOR_OPART].SectorSpansBoundary			:= FALSE; 	
	
	SectorConfig[GC.SHORTCUT_ENTRY_SECTOR_IPART].PartObjectId					:= GVL_General.XtsPartInnerFinish;
	SectorConfig[GC.SHORTCUT_ENTRY_SECTOR_IPART].PartSectorStartPosn			:= 0;
	SectorConfig[GC.SHORTCUT_ENTRY_SECTOR_IPART].PartSectorEndPosn			:= stTrackGlobalConfig.ShortcutShuttleFullyInPosn;
	SectorConfig[GC.SHORTCUT_ENTRY_SECTOR_IPART].TrackSectorStartPosn		:= 0;
	SectorConfig[GC.SHORTCUT_ENTRY_SECTOR_IPART].TrackSectorEndPosn 			:= 0;

	SectorConfig[GC.SHORTCUT_ENTRY_HALF_IPART].PartObjectId						:= GVL_General.XtsPartInnerFinish;
	SectorConfig[GC.SHORTCUT_ENTRY_HALF_IPART].PartSectorStartPosn			:= 0;
	SectorConfig[GC.SHORTCUT_ENTRY_HALF_IPART].PartSectorEndPosn			 	:= (GVL_Mc3.MC_Tracks[E_TrackNum.Small].GetLength() / 2);
	SectorConfig[GC.SHORTCUT_ENTRY_HALF_IPART].TrackSectorStartPosn			:= 0;
	SectorConfig[GC.SHORTCUT_ENTRY_HALF_IPART].TrackSectorEndPosn 			:= 0;

	SectorConfig[GC.SHORTCUT_CALC_SECTOR_IPART].PartObjectId						:= GVL_General.XtsPartInnerFinish;
	SectorConfig[GC.SHORTCUT_CALC_SECTOR_IPART].PartSectorStartPosn			:= 0;
	SectorConfig[GC.SHORTCUT_CALC_SECTOR_IPART].PartSectorEndPosn			:= GVL_Mc3.MC_Tracks[E_TrackNum.Small].GetLength()-stTrackGlobalConfig.MergeWaitFinishDistance + (stMoverConfig.NormalMoverGap /2);
	SectorConfig[GC.SHORTCUT_CALC_SECTOR_IPART].TrackSectorStartPosn			:= 0;
	SectorConfig[GC.SHORTCUT_CALC_SECTOR_IPART].TrackSectorEndPosn 			:= 0;

	SectorConfig[GC.LOAD_STOP_SECTOR_IPART].PartObjectId						    := GVL_General.XtsPartInnerFinish;
	SectorConfig[GC.LOAD_STOP_SECTOR_IPART].PartSectorStartPosn			    := F_PosnInitial(VeloInit := GVL_General.stMoverConfig.NormalVelo, VeloFinal := 0, Accel := GVL_General.stMoverConfig.NormalDecel, PosnFinal := (GVL_Mc3.MC_Tracks[E_TrackNum.Small].GetLength() /2) -GC.SHUTTLE_LENGTH);
	SectorConfig[GC.LOAD_STOP_SECTOR_IPART].PartSectorEndPosn			 	:= GC.SHUTTLE_LENGTH + (GVL_Mc3.MC_Tracks[E_TrackNum.Small].GetLength() /2) ;
	SectorConfig[GC.LOAD_STOP_SECTOR_IPART].TrackSectorStartPosn			    := 0;
	SectorConfig[GC.LOAD_STOP_SECTOR_IPART].TrackSectorEndPosn 			 	:= 0;

	SectorConfig[GC.SHORTCUT_COMPLETE].PartObjectId													:= GVL_General.XtsPartInnerFinish;
	SectorConfig[GC.SHORTCUT_COMPLETE].PartSectorStartPosn								:= 0;
	SectorConfig[GC.SHORTCUT_COMPLETE].PartSectorEndPosn								:= GVL_Mc3.MC_Tracks[E_TrackNum.Small].GetLength();
	SectorConfig[GC.SHORTCUT_COMPLETE].TrackSectorStartPosn						:= 0;
	SectorConfig[GC.SHORTCUT_COMPLETE].TrackSectorEndPosn 							:= 0;
	
	SectorConfig[GC.SHORTCUT_HD_SECTION].PartObjectId										:= GVL_General.XtsPartInnerFinish;
	SectorConfig[GC.SHORTCUT_HD_SECTION].PartSectorStartPosn							:= stTrackGlobalConfig.ShortcutHDRegionDistance;
	SectorConfig[GC.SHORTCUT_HD_SECTION].PartSectorEndPosn								:= GVL_Mc3.MC_Tracks[E_TrackNum.Small].GetLength()-stTrackGlobalConfig.ShortcutHDRegionDistance;
	SectorConfig[GC.SHORTCUT_HD_SECTION].TrackSectorStartPosn						:= 0;
	SectorConfig[GC.SHORTCUT_HD_SECTION].TrackSectorEndPosn 							:= 0;
	
	SectorConfig[GC.SHORTCUT_EXIT_HALF_IPART].PartObjectId										:= GVL_General.XtsPartInnerFinish;
	SectorConfig[GC.SHORTCUT_EXIT_HALF_IPART].PartSectorStartPosn				:= (GVL_Mc3.MC_Tracks[E_TrackNum.Small].GetLength() / 2);
	SectorConfig[GC.SHORTCUT_EXIT_HALF_IPART].PartSectorEndPosn			 		:= GVL_Mc3.MC_Tracks[E_TrackNum.Small].GetLength();
	SectorConfig[GC.SHORTCUT_EXIT_HALF_IPART].TrackSectorStartPosn				:= 0;
	SectorConfig[GC.SHORTCUT_EXIT_HALF_IPART].TrackSectorEndPosn 				:= 0;

	SectorConfig[GC.SHORTCUT_MERGE_COMMAND_WAIT].PartObjectId								:= GVL_General.XtsPartInnerFinish;
	SectorConfig[GC.SHORTCUT_MERGE_COMMAND_WAIT].PartSectorStartPosn					:= F_PosnInitial(VeloInit := GVL_General.stMoverConfig.NormalVelo, VeloFinal := 0, Accel := GVL_General.stMoverConfig.NormalDecel, PosnFinal := (GVL_Mc3.MC_Tracks[E_TrackNum.Small].GetLength()-stTrackGlobalConfig.MergeWaitFinishDistance-stTrackGlobalConfig.MergeWaitAccelDistance));
	SectorConfig[GC.SHORTCUT_MERGE_COMMAND_WAIT].PartSectorEndPosn						:= GVL_Mc3.MC_Tracks[E_TrackNum.Small].GetLength()-stTrackGlobalConfig.MergeWaitFinishDistance + (GC.SHUTTLE_LENGTH /2);
	SectorConfig[GC.SHORTCUT_MERGE_COMMAND_WAIT].TrackSectorStartPosn					:= 0;
	SectorConfig[GC.SHORTCUT_MERGE_COMMAND_WAIT].TrackSectorEndPosn 					:= 0;
	
	SectorConfig[GC.SHORTCUT_MERGE_COMMAND_FLYING].PartObjectId								:= GVL_General.XtsPartInnerFinish;
	SectorConfig[GC.SHORTCUT_MERGE_COMMAND_FLYING].PartSectorStartPosn					:= SectorConfig[GC.SHORTCUT_MERGE_COMMAND_WAIT].PartSectorStartPosn - GC.SHUTTLE_LENGTH;
	SectorConfig[GC.SHORTCUT_MERGE_COMMAND_FLYING].PartSectorEndPosn						:= SectorConfig[GC.SHORTCUT_MERGE_COMMAND_WAIT].PartSectorStartPosn;
	SectorConfig[GC.SHORTCUT_MERGE_COMMAND_FLYING].TrackSectorStartPosn				:= 0;
	SectorConfig[GC.SHORTCUT_MERGE_COMMAND_FLYING].TrackSectorEndPosn 					:= 0;

	//for calculation of length in the "3rd condition"
	SectorConfig[GC.SHORTCUT_MERGE_CALC_EXACT].PartObjectId										:= GVL_General.XtsPartInnerFinish;
	SectorConfig[GC.SHORTCUT_MERGE_CALC_EXACT].PartSectorStartPosn					:= F_PosnInitial(VeloInit := GVL_General.stMoverConfig.NormalVelo, VeloFinal := 0, Accel := GVL_General.stMoverConfig.NormalDecel, PosnFinal := (GVL_Mc3.MC_Tracks[E_TrackNum.Small].GetLength()-stTrackGlobalConfig.MergeWaitFinishDistance));
	SectorConfig[GC.SHORTCUT_MERGE_CALC_EXACT].PartSectorEndPosn						:= GVL_Mc3.MC_Tracks[E_TrackNum.Small].GetLength()-stTrackGlobalConfig.MergeWaitFinishDistance;
	SectorConfig[GC.SHORTCUT_MERGE_CALC_EXACT].TrackSectorStartPosn					:= 0;
	SectorConfig[GC.SHORTCUT_MERGE_CALC_EXACT].TrackSectorEndPosn 					:= 0;
	
	SectorConfig[GC.INNER_MERGE_TO_FINISH].PartObjectId						   				 := GVL_General.XtsPartInnerFinish;
	SectorConfig[GC.INNER_MERGE_TO_FINISH].PartSectorStartPosn					    := F_PosnInitial(VeloInit := GVL_General.stMoverConfig.NormalVelo, VeloFinal := 0, Accel := GVL_General.stMoverConfig.NormalDecel, PosnFinal := GVL_Mc3.MC_Tracks[E_TrackNum.Small].GetLength());
	SectorConfig[GC.INNER_MERGE_TO_FINISH].PartSectorEndPosn			 				:= GVL_Mc3.MC_Tracks[E_TrackNum.Small].GetLength();
	SectorConfig[GC.INNER_MERGE_TO_FINISH].TrackSectorStartPosn					   	:= 0;
	SectorConfig[GC.INNER_MERGE_TO_FINISH].TrackSectorEndPosn 					 	:= 0;
                                                                            
	SectorConfig[GC.OUTER_MERGE_COLLISION].PartObjectId						 	 					:= GVL_General.XtsPartOuterFinish;
	SectorConfig[GC.OUTER_MERGE_COLLISION].PartSectorStartPosn			 	 				:= F_PosnInitial(VeloInit := GVL_General.stMoverConfig.NormalVelo, VeloFinal := 0, Accel := GVL_General.stMoverConfig.NormalDecel, PosnFinal := (GVL_Mc3.MC_Tracks[E_TrackNum.Big].GetLength() - stTrackGlobalConfig.MergeCollisionRegionDeltaFromL));
	SectorConfig[GC.OUTER_MERGE_COLLISION].PartSectorEndPosn			 	 	 				:= GVL_Mc3.MC_Tracks[E_TrackNum.Big].GetLength() - stTrackGlobalConfig.MergeCollisionAdvance;
	SectorConfig[GC.OUTER_MERGE_COLLISION].TrackSectorStartPosn			 				:= 0;
	SectorConfig[GC.OUTER_MERGE_COLLISION].TrackSectorEndPosn 			 					:= 0;
	SectorConfig[GC.OUTER_MERGE_COLLISION].SectorSpansBoundary 			 				:= FALSE;
	
	SectorConfig[GC.OUTER_SHORTCUT_PROJECTIONFLY].PartObjectId						 	 		:= GVL_General.XtsPartOuterFinish;
	SectorConfig[GC.OUTER_SHORTCUT_PROJECTIONFLY].PartSectorStartPosn			 	 	:= GVL_Mc3.MC_Tracks[E_TrackNum.Big].GetLength() - SectorConfig[GC.SHORTCUT_MERGE_COMMAND_WAIT].PartSectorStartPosn - stTrackGlobalConfig.ExpMoverLength;
	SectorConfig[GC.OUTER_SHORTCUT_PROJECTIONFLY].PartSectorEndPosn			 	 	 	:= GVL_Mc3.MC_Tracks[E_TrackNum.Big].GetLength() - SectorConfig[GC.SHORTCUT_MERGE_COMMAND_WAIT].PartSectorStartPosn;
	SectorConfig[GC.OUTER_SHORTCUT_PROJECTIONFLY].TrackSectorStartPosn			 	:= 0;
	SectorConfig[GC.OUTER_SHORTCUT_PROJECTIONFLY].TrackSectorEndPosn 			 			:= 0;
	SectorConfig[GC.OUTER_SHORTCUT_PROJECTIONFLY].SectorSpansBoundary 			 	:= FALSE;
	
	SectorConfig[GC.OUTER_SHORTCUT_PROJECTIONSTAT].PartObjectId						 	 		:= GVL_General.XtsPartOuterFinish;
	SectorConfig[GC.OUTER_SHORTCUT_PROJECTIONSTAT].PartSectorStartPosn			 	 	:= GVL_Mc3.MC_Tracks[E_TrackNum.Small].GetLength() - stTrackGlobalConfig.MergeWaitFinishDistance - stTrackGlobalConfig.ExpMoverLength;
	SectorConfig[GC.OUTER_SHORTCUT_PROJECTIONSTAT].PartSectorEndPosn			 	 	 	:= GVL_Mc3.MC_Tracks[E_TrackNum.Small].GetLength() - stTrackGlobalConfig.MergeWaitFinishDistance; (*-stTrackGlobalConfig.MergeWaitAccelDistance*)
	SectorConfig[GC.OUTER_SHORTCUT_PROJECTIONSTAT].TrackSectorStartPosn			 	:= 0;
	SectorConfig[GC.OUTER_SHORTCUT_PROJECTIONSTAT].TrackSectorEndPosn 			 			:= 0;
	SectorConfig[GC.OUTER_SHORTCUT_PROJECTIONSTAT].SectorSpansBoundary 			 	:= FALSE;
	
//Multi
	SectorConfig[GC.OUTER_TIGHTGAP_ZONE].PartObjectIdEnt						 	:= GVL_General.XtsPartOuterFinish;
	SectorConfig[GC.OUTER_TIGHTGAP_ZONE].PartObjectIdExit						 	:= GVL_General.XtsPartOuterStart;
	SectorConfig[GC.OUTER_TIGHTGAP_ZONE].PartSectorStartPosn			 	 		:= GVL_Mc3.MC_Tracks[E_TrackNum.Big].GetLength() - stMoverConfig.NormalMoverGap; // take the distance from the small track 
	SectorConfig[GC.OUTER_TIGHTGAP_ZONE].PartSectorEndPosn			 	 	 		:= stMoverConfig.NormalMoverGap;
	SectorConfig[GC.OUTER_TIGHTGAP_ZONE].TrackSectorStartPosn			 		:= 0;//GVL_Mc3.MC_Tracks[E_TrackNum.Main].GetLength() + astSectorConfig[GC.OUTER_MERGE_FINISH].PartSectorStartPosn;
	SectorConfig[GC.OUTER_TIGHTGAP_ZONE].TrackSectorEndPosn 			 			:= 0;//astSectorConfig[GC.OUTER_MERGE_START].PartSectorEndPosn;
	SectorConfig[GC.OUTER_TIGHTGAP_ZONE].SectorSpansBoundary					:= TRUE;
	
	SectorConfig[GC.OUTER_PRE_TG_ZONE].PartObjectId						 	 			:= GVL_General.XtsPartOuterFinish;
	SectorConfig[GC.OUTER_PRE_TG_ZONE].PartSectorStartPosn			 	 		:= SectorConfig[GC.OUTER_TIGHTGAP_ZONE].PartSectorStartPosn - stMoverConfig.NormalMoverGap;
	SectorConfig[GC.OUTER_PRE_TG_ZONE].PartSectorEndPosn			 	 	 		:= SectorConfig[GC.OUTER_TIGHTGAP_ZONE].PartSectorStartPosn;
	SectorConfig[GC.OUTER_PRE_TG_ZONE].TrackSectorStartPosn			 			:= 0;
	SectorConfig[GC.OUTER_PRE_TG_ZONE].TrackSectorEndPosn 			 				:= 0;
	SectorConfig[GC.OUTER_PRE_TG_ZONE].SectorSpansBoundary					:= FALSE;
	
	SectorConfig[GC.OUTER_POST_TG_ZONE].PartObjectId						 	 			:= GVL_General.XtsPartOuterStart;
	SectorConfig[GC.OUTER_POST_TG_ZONE].PartSectorStartPosn			 	 		:= SectorConfig[GC.OUTER_TIGHTGAP_ZONE].PartSectorEndPosn;
	SectorConfig[GC.OUTER_POST_TG_ZONE].PartSectorEndPosn			 	 	 		:= SectorConfig[GC.OUTER_TIGHTGAP_ZONE].PartSectorEndPosn + stMoverConfig.NormalMoverGap;
	SectorConfig[GC.OUTER_POST_TG_ZONE].TrackSectorStartPosn			 			:= 0;
	SectorConfig[GC.OUTER_POST_TG_ZONE].TrackSectorEndPosn 			 				:= 0;
	SectorConfig[GC.OUTER_POST_TG_ZONE].SectorSpansBoundary					:= FALSE;

	SectorConfig[GC.OUTER_BIGTRACK_END].PartObjectId						 	 					:= GVL_General.XtsPartOuterFinish;
	SectorConfig[GC.OUTER_BIGTRACK_END].PartSectorStartPosn			 	 		:= F_PosnInitial(VeloInit := GVL_General.stMoverConfig.NormalVelo, VeloFinal := 0, Accel := GVL_General.stMoverConfig.NormalDecel, PosnFinal := GVL_Mc3.MC_Tracks[E_TrackNum.Big].GetLength()) - GC.SHUTTLE_LENGTH;
	SectorConfig[GC.OUTER_BIGTRACK_END].PartSectorEndPosn			 	 	 		:= GVL_Mc3.MC_Tracks[E_TrackNum.Big].GetLength();
	SectorConfig[GC.OUTER_BIGTRACK_END].TrackSectorStartPosn			 			:= 0;
	SectorConfig[GC.OUTER_BIGTRACK_END].TrackSectorEndPosn 			 				:= 0;
	SectorConfig[GC.OUTER_BIGTRACK_END].SectorSpansBoundary					:= FALSE;
	
	SectorConfig[GC.OUTER_BIGTRACK_LSMALL].PartObjectId						 	 			:= GVL_General.XtsPartOuterFinish;
	SectorConfig[GC.OUTER_BIGTRACK_LSMALL].PartSectorStartPosn			 	 		:= GVL_Mc3.MC_Tracks[E_TrackNum.Big].GetLength() - GVL_Mc3.MC_Tracks[E_TrackNum.Small].GetLength();
	SectorConfig[GC.OUTER_BIGTRACK_LSMALL].PartSectorEndPosn			 	 	 		:= GVL_Mc3.MC_Tracks[E_TrackNum.Big].GetLength();
	SectorConfig[GC.OUTER_BIGTRACK_LSMALL].TrackSectorStartPosn			 			:= GVL_Mc3.MC_Tracks[E_TrackNum.Big].GetLength() - GVL_Mc3.MC_Tracks[E_TrackNum.Small].GetLength();
	SectorConfig[GC.OUTER_BIGTRACK_LSMALL].TrackSectorEndPosn 			 				:= GVL_Mc3.MC_Tracks[E_TrackNum.Big].GetLength();                                                
	SectorConfig[GC.OUTER_BIGTRACK_LSMALL].SectorSpansBoundary					:= FALSE;

	SectorConfig[GC.OUTER_BIGTRACK_MOVE_END].PartObjectId						 	 		:= GVL_General.XtsPartOuterFinish;
	SectorConfig[GC.OUTER_BIGTRACK_MOVE_END].PartSectorStartPosn			 	 		:= GVL_Mc3.MC_Tracks[E_TrackNum.Big].GetLength() - stTrackGlobalConfig.TargetPosnBeforeTrackEnd;
	SectorConfig[GC.OUTER_BIGTRACK_MOVE_END].PartSectorEndPosn			 	 	 		:= GVL_Mc3.MC_Tracks[E_TrackNum.Big].GetLength();
	SectorConfig[GC.OUTER_BIGTRACK_MOVE_END].TrackSectorStartPosn			 			:= 0;
	SectorConfig[GC.OUTER_BIGTRACK_MOVE_END].TrackSectorEndPosn 			 				:= 0;
	SectorConfig[GC.OUTER_BIGTRACK_MOVE_END].SectorSpansBoundary					:= FALSE;
END_IF
END_METHOD

METHOD PRIVATE _M_UpdateMultiSectors
//Update Multi Sectors

//MergeCombinedSectorStat.MoverCountOnSector			:= afbSector[GC.OUTER_MERGE_START].P_SectorStatus.MoverCountOnSector + 
//                                                  afbSector[GC.OUTER_MERGE_FINISH].P_SectorStatus.MoverCountOnSector;
																									
//MergeCombinedSectorStat.MoverIsOnSector				:= NOT (MergeCombinedSectorStat.MoverCountOnSector = 0);
END_METHOD

METHOD PROTECTED _M_UpdateStatus
VAR
    SectorIndex : INT; // FOR loop
END_VAR
//Update Singular Sectors
FOR SectorIndex := GC.MIN_SECTOR_CT TO GC.MAX_SECTOR_CT DO
    IF afbSector[SectorIndex].P_SectorStatus.MoverEnteredSector.Q THEN
        afbSector[SectorIndex].P_SectorStatus.MoverCountOnSector	:= afbSector[SectorIndex].P_SectorStatus.MoverCountOnSector +1;
				LinkedMoveList[SectorIndex].AddObjToBuffer(RefObject := iMover);
    ELSIF afbSector[SectorIndex].P_SectorStatus.MoverExitedSector.Q THEN
        afbSector[SectorIndex].P_SectorStatus.MoverCountOnSector	:= afbSector[SectorIndex].P_SectorStatus.MoverCountOnSector -1;
				LinkedMoveList[SectorIndex].RemoveObjFromBuffer();
    END_IF
		
		SectorStatus[SectorIndex]										:=  afbSector[SectorIndex].P_SectorStatus;
END_FOR
END_METHOD

//FB_Init is always available implicitly and it is used primarily for initialization.
//The return value is not evaluated. For a specific influence, you can also declare the
//methods explicitly and provide additional code there with the standard initialization
//code. You can evaluate the return value.
METHOD FB_Init: BOOL
VAR_INPUT
    bInitRetains: BOOL; // TRUE: the retain variables are initialized (reset warm / reset cold)
    bInCopyCode: BOOL;  // TRUE: the instance will be copied to the copy code afterward (online change)   
END_VAR
SectorsConfig.AllSectorsConfig	REF= SectorConfig;
SectorsStatus.AllSectorsStatus		REF= SectorStatus;
END_METHOD

PROPERTY P_SectorsConfig : REFERENCE TO ST_SectorsConfig
GET
P_SectorsConfig REF= SectorsConfig;
END_GET
END_PROPERTY

PROPERTY P_SectorsStatus : REFERENCE TO ST_SectorsStatus
GET
P_SectorsStatus REF= SectorsStatus;
END_GET
END_PROPERTY

END_FUNCTION_BLOCK

// ---- POUs/FBs/FB_TrackSector.TcPOU
FUNCTION_BLOCK FB_TrackSector
VAR_INPUT
	PlanarTrackIndex				: E_TrackNum := E_TrackNum.Small;
END_VAR
VAR_IN_OUT
	refPlanarTracks					: ARRAY[*] OF ST_PlanarTrackConfig; //NOTE ref array is 0-based!
END_VAR                     		
VAR                             	
	InitDone						: BOOL;
	stSectorConfig					: ST_SectorConfig;
	LowerBoundPlanarTrackConfig		: DINT;
	UpperBoundPlanarTrackConfig		: DINT;
	refXtsMover						: Tc3_XTS_Utility.ST_PositionInfo;
	refPlanarMover					: MoverSort;
	stSectorStatus				: ST_SectorStatus;
END_VAR

IF UpperBoundPlanarTrackConfig = 0 THEN
	_M_Init();
ELSE
	InitDone	:= TRUE;
END_IF

IF InitDone THEN
	_M_UpdateSectorStatus();
END_IF

METHOD PROTECTED _M_EnteredSectorBoundary : BOOL
//By XTS Loop
_M_EnteredSectorBoundary	:= ((refXtsMover.nTrackObjectid = stSectorConfig.TrackObjectId) OR
											(refXtsMover.nPartObjectid = stSectorConfig.PartObjectIdEnt)) AND
											(refXtsMover.fPartPosition >= stSectorConfig.PartSectorStartPosn);
END_METHOD

METHOD PROTECTED _M_ExitedSectorBoundary : BOOL
//By XTS Loop
_M_ExitedSectorBoundary	:= ((refXtsMover.nTrackObjectid = stSectorConfig.TrackObjectId) OR
											(refXtsMover.nPartObjectid = stSectorConfig.PartObjectIdExit)) AND 		
											(refXtsMover.fPartPosition > stSectorConfig.PartSectorEndPosn);
END_METHOD

METHOD PRIVATE _M_Init
LowerBoundPlanarTrackConfig	:= LOWER_BOUND(refPlanarTracks,1);
UpperBoundPlanarTrackConfig	:= UPPER_BOUND(refPlanarTracks,1);
END_METHOD

METHOD PROTECTED _M_IsOnBoundarySector
VAR_INST
	MoverEnteredOneShot 	: BOOL;
	MoverExitedOneShot	: BOOL;
END_VAR
//By XTS Loop
IF NOT MoverEnteredOneShot AND _M_EnteredSectorBoundary() THEN
	stSectorStatus.MoverIsOnSector	:= TRUE;
	MoverEnteredOneShot	:= TRUE;
END_IF

IF MoverEnteredOneShot THEN
	IF NOT MoverExitedOneShot AND _M_ExitedSectorBoundary() THEN
		stSectorStatus.MoverIsOnSector	:= FALSE;
		MoverExitedOneShot := TRUE;
	END_IF
END_IF

IF stSectorStatus.MoverExitedSector.Q THEN
	MoverEnteredOneShot 	:= FALSE;
	MoverExitedOneShot		:= FALSE;
END_IF
END_METHOD

METHOD PROTECTED _M_IsOnPlanarSector : BOOL
//note refPlanarTracks ARRAY is 0-based!
IF ADR(refPlanarTracks[(PlanarTrackIndex-1)]) <> 0 THEN
	_M_IsOnPlanarSector	:= (refPlanarMover.TrackID = refPlanarTracks[(PlanarTrackIndex-1)].MCTrack.TrackOID) 
							AND IsBetween(value := refPlanarMover.MoverPos, 
												minV := stSectorConfig.TrackSectorStartPosn, 
												maxV := stSectorConfig.TrackSectorEndPosn);
END_IF
END_METHOD

METHOD PROTECTED _M_IsOnXtsSector : BOOL
//By XTS Loop
_M_IsOnXtsSector	:= ((refXtsMover.nTrackObjectid = stSectorConfig.TrackObjectId) OR
										(refXtsMover.nPartObjectid = stSectorConfig.PartObjectId)) AND
										(IsBetween(value := refXtsMover.fPartPosition, 
										minV := stSectorConfig.PartSectorStartPosn, 
										maxV := stSectorConfig.PartSectorEndPosn) OR
										IsBetween(value := refXtsMover.fTrackPosition, 
										minV := stSectorConfig.TrackSectorStartPosn, 
										maxV := stSectorConfig.TrackSectorEndPosn));
END_METHOD

METHOD PROTECTED _M_UpdateSectorStatus
IF stSectorConfig.SectorSpansBoundary THEN
	_M_IsOnBoundarySector();
ELSE // by parts
	stSectorStatus.MoverIsOnSector	:= _M_IsOnXtsSector() ; //OR _M_IsOnPlanarSector(); this method works, but I believe the reference VAR_IN_OUT type is causing problems (duplication) here
END_IF

stSectorStatus.MoverEnteredSector(CLK := stSectorStatus.MoverIsOnSector);
stSectorStatus.MoverExitedSector(CLK := stSectorStatus.MoverIsOnSector);

stSectorStatus.SectorLength := stSectorConfig.PartSectorEndPosn - stSectorConfig.PartSectorStartPosn;

IF stSectorStatus.MoverIsOnSector THEN
	stSectorStatus.MoverDistanceFromEnd := stSectorConfig.PartSectorEndPosn - refXtsMover.fPartPosition;
ELSE
	stSectorStatus.MoverDistanceFromEnd	:= 0;
END_IF

IF stSectorStatus.MoverIsOnSector THEN
	IF stSectorStatus.SectorLength <> 0 THEN
		stSectorStatus.PercentOfSectorTraversed	:= (refXtsMover.fPartPosition - stSectorConfig.PartSectorStartPosn) / stSectorStatus.SectorLength;
	END_IF
END_IF
END_METHOD

PROPERTY P_MoverSort : REFERENCE TO MoverSort
GET
P_MoverSort	REF= refPlanarMover;
END_GET
END_PROPERTY

PROPERTY P_SectorStatus : REFERENCE TO ST_SectorStatus
GET
P_SectorStatus	REF= stSectorStatus;
END_GET
END_PROPERTY

PROPERTY P_TrackSectorConfig : REFERENCE TO ST_SectorConfig
GET
P_TrackSectorConfig REF= stSectorConfig;
END_GET
END_PROPERTY

PROPERTY P_XtsPositionInfo : REFERENCE TO Tc3_XTS_Utility.ST_PositionInfo
GET
P_XtsPositionInfo REF= refXtsMover;
END_GET
END_PROPERTY

END_FUNCTION_BLOCK

// ---- POUs/FUNs/F_PosnInitial.TcPOU
FUNCTION F_PosnInitial : LREAL
VAR_INPUT
	VeloInit 	: LREAL;
	VeloFinal	: LREAL;
	Accel		: LREAL;
	PosnFinal	: LREAL;
END_VAR
VAR
END_VAR

IF ((2*Accel) + PosnFinal) <> 0 THEN
	F_PosnInitial := ((EXPT(VeloFinal,2) - EXPT(VeloInit,2)) / (2*Accel)) + PosnFinal;
END_IF

END_FUNCTION

// ---- POUs/FBs/FB_AllTrackSectors.TcPOU
FUNCTION_BLOCK FB_AllTrackSectors
VAR_INPUT
	TrackSectorsRef				: REFERENCE TO ARRAY[GC.nNumMinMovers..GC.nNumMaxMovers] OF FB_TrackSectors;
	HeadTrackSectorsRef		: REFERENCE TO ARRAY[GC.nNumMinMovers..GC.nNumMaxMovers] OF FB_TrackSectors;
	TailTrackSectorsRef		: REFERENCE TO ARRAY[GC.nNumMinMovers..GC.nNumMaxMovers] OF FB_TrackSectors;		
END_VAR
//VAR_IN_OUT CONSTANT //not writeable by this FB
//		TrackSectorsRef				: ARRAY[*] OF FB_TrackSectors;
//END_VAR
VAR
	iSectors				: ARRAY[GC.nNumMinMovers..GC.nNumMaxMovers] OF I_MoverSector;
	DynamicMergeEvaluation : BOOL;
	MoverIndex			: UDINT;
	ForCounterExit : ARRAY[GC.MIN_TRACKSECTORS_REF..GC.MAX_TRACKSECTORS_REF] OF ARRAY[GC.MIN_SECTOR_CT..GC.MAX_SECTOR_CT] OF UDINT; // 1 to 3 are normal, Head, Tail TrackSectorsRef
	ForCounterDuringClear : UDINT;
	SectorIndex : UDINT;
	AllRealSectorStatus	: ARRAY[GC.nNumMinMovers..GC.nNumMaxMovers] OF ARRAY[GC.MIN_SECTOR_CT..GC.MAX_SECTOR_CT] OF ST_SectorStatus;
	AllHeadSectorStatus : ARRAY[GC.nNumMinMovers..GC.nNumMaxMovers] OF ARRAY[GC.MIN_SECTOR_CT..GC.MAX_SECTOR_CT] OF ST_SectorStatus;
	AllTailSectorStatus : ARRAY[GC.nNumMinMovers..GC.nNumMaxMovers] OF ARRAY[GC.MIN_SECTOR_CT..GC.MAX_SECTOR_CT] OF ST_SectorStatus;
	LowerOut : DINT;
	UpperOut : DINT;
	RealMoverIsOnSector	: ARRAY[GC.MIN_SECTOR_CT..GC.MAX_SECTOR_CT] OF BOOL;
	ValidMerge				: RingBuffer.ST_MoverMerge;
	TempWindowStartPosn		: LREAL;
	MoverIdMergeOnSector		: UDINT;
	MoverInDecelSector			: BOOL;
	TimeForShortcutMergingMover : LREAL;
	ValidMergeTrig				: BOOL;
	ClearZone				: BOOL;
END_VAR

//LowerOut := LOWER_BOUND(TrackSectorsRef, 1);
//UpperOut := UPPER_BOUND(TrackSectorsRef, 1);

//IF LowerOut<>0 AND UpperOut<>0 THEN
	_M_EvaluateStatus();
//END_IF

METHOD PROTECTED _M_BufferValidMergeRefs
VAR_INST
	RealMoverEnteredSector : Tc2_Standard.R_TRIG;
END_VAR
//Do FOR loop for all of the sectors later
_M_IsRealMoverOnSector(SectorID := GC.OUTER_SHORTCUT_PROJECTIONFLY);
_M_IsRealMoverOnSector(SectorID := GC.OUTER_BIGTRACK_LSMALL);


//Checking Expanded Movers against real mover locations
FOR ForCounterExit[GC.TRACK_SECTORS_HEAD][GC.OUTER_SHORTCUT_PROJECTIONFLY] := GC.nNumMinMovers TO GC.nNumMaxMovers DO
	IF NOT RealMoverIsOnSector[GC.OUTER_SHORTCUT_PROJECTIONFLY] THEN
		IF HeadTrackSectorsRef[ForCounterExit[GC.TRACK_SECTORS_HEAD][GC.OUTER_SHORTCUT_PROJECTIONFLY]].SectorStatus[GC.OUTER_SHORTCUT_PROJECTIONFLY].MoverEnteredSector.Q AND NOT ClearZone THEN 
			ValidMerge.MoverID 			:= ForCounterExit[GC.TRACK_SECTORS_HEAD][GC.OUTER_SHORTCUT_PROJECTIONFLY];
			ValidMerge.ExpMoverType 	:= E_ExpMover.Head;
			ValidMerge.MergeWindowStartPosn	:= HeadExpMover[ValidMerge.MoverID].P_ExpMoverStatus.XtsAdjustedData.fPartPosition;
			ClearZone	 := TRUE;
			EXIT;
		END_IF
	END_IF
END_FOR

FOR ForCounterDuringClear := GC.nNumMinMovers TO GC.nNumMaxMovers DO
	IF ValidMerge.MoverID <> 0 THEN
		
		IF ClearZone AND HeadTrackSectorsRef[ValidMerge.MoverID].SectorStatus[GC.OUTER_SHORTCUT_PROJECTIONFLY].MoverExitedSector.Q THEN
			ValidMerge.MergeWindowEndPosn	:= HeadExpMover[ValidMerge.MoverID].P_ExpMoverStatus.XtsAdjustedData.fPartPosition;
			ValidMergeTrig := TRUE;
		ELSIF RealMoverIsOnSector[GC.OUTER_SHORTCUT_PROJECTIONFLY] THEN
			ClearZone 	:= FALSE;
		END_IF
		
	END_IF
END_FOR

IF ValidMergeTrig AND ValidMerge.MergeWindowStartPosn <> TempWindowStartPosn THEN
	MergeQueue.AddObjToBuffer(RefObject := ValidMerge);
	TempWindowStartPosn	:= ValidMerge.MergeWindowStartPosn;
	ValidMergeTrig	:= FALSE;
END_IF

//Delete queue objects when they reach the merge position
IF MergeQueue.P_LastObjectRemoved.MoverID <> 0 THEN
	IF HeadTrackSectorsRef[MergeQueue.P_LastObjectRemoved.MoverID].SectorStatus[GC.OUTER_BIGTRACK_MOVE_END].MoverEnteredSector.Q THEN
//		MergeQueue.ClearLastRemoved();
	END_IF
END_IF

RealMoverEnteredSector(CLK := RealMoverIsOnSector[GC.OUTER_SHORTCUT_PROJECTIONFLY]);
END_METHOD

METHOD _M_CalculateTCompForMerge
//Calculate t if mover is between the start and end of this sector; this t is used to relate the constant velocity region on the outer loop
IF MoverIdMergeOnSector <> 0 THEN
	IF TrackSectorsRef[MoverIdMergeOnSector].SectorStatus[GC.SHORTCUT_MERGE_CALC_EXACT].MoverIsOnSector AND MoverInDecelSector THEN
		//This is only calculated for one mover at once
		TimeForShortcutMergingMover := F_t_SL2a(SectorLength := TrackSectorsRef[MoverIdMergeOnSector].SectorStatus[GC.SHORTCUT_MERGE_CALC_EXACT].MoverDistanceFromEnd, 
																						Acceleration := stMoverConfig.MaxDecel);
	END_IF
	
	IF TrackSectorsRef[MoverIdMergeOnSector].SectorStatus[GC.SHORTCUT_MERGE_CALC_EXACT].MoverExitedSector.Q AND MoverInDecelSector THEN
		MoverInDecelSector		:= FALSE;
	END_IF
END_IF
END_METHOD

METHOD PRIVATE _M_EvaluateStatus
IF ADR(TrackSectorsRef) <> 0 THEN // pointer validity check
	FOR MoverIndex := GC.nNumMinMovers TO GVL_General.nNumMovers BY 1 DO
		
		iSectors[MoverIndex]	:= TrackSectorsRef[MoverIndex];
		
	//Write All Sector Status
		FOR SectorIndex := GC.MIN_SECTOR_CT TO GC.MAX_SECTOR_CT BY 1 DO
			//Note!: VAR_IN_OUT (REF) Arrays are O-Based! 
			AllRealSectorStatus[MoverIndex][SectorIndex] := TrackSectorsRef[(MoverIndex)].SectorStatus[(SectorIndex)];
			AllHeadSectorStatus[MoverIndex][SectorIndex] := HeadTrackSectorsRef[(MoverIndex)].SectorStatus[(SectorIndex)];
			AllTailSectorStatus[MoverIndex][SectorIndex] := TailTrackSectorsRef[(MoverIndex)].SectorStatus[(SectorIndex)];
		END_FOR

		IF TrackSectorsRef[MoverIndex].SectorStatus[GC.SHORTCUT_MERGE_CALC_EXACT].MoverEnteredSector.Q AND NOT MoverInDecelSector THEN
			MoverIdMergeOnSector 	:= MoverIndex;
			MoverInDecelSector		:= TRUE;
		END_IF

	END_FOR
END_IF

IF NOT DynamicMergeEvaluation THEN
	_M_StaticSectorClear();
ELSE
	// // ELSIF Config.UseExpandedMovers
END_IF

//Do all this
_M_CalculateTCompForMerge();

_M_BufferValidMergeRefs();
END_METHOD

METHOD PRIVATE _M_IsRealMoverOnSector
VAR_INPUT
	SectorID : UDINT;
END_VAR
//Merge - 'If Any'
FOR ForCounterExit[GC.TRACK_SECTORS_STD][SectorID] := GC.nNumMinMovers TO GVL_General.nNumMovers BY 1 DO
	IF AllRealSectorStatus[ForCounterExit[GC.TRACK_SECTORS_STD][SectorID]][SectorID].MoverIsOnSector THEN
			RealMoverIsOnSector[SectorID] := TRUE;
			EXIT;
		ELSIF NOT AllRealSectorStatus[ForCounterExit[GC.TRACK_SECTORS_STD][SectorID]][SectorID].MoverIsOnSector THEN
			RealMoverIsOnSector[SectorID] := FALSE;
		END_IF
	
END_FOR
END_METHOD

METHOD PRIVATE _M_StaticSectorClear
//Checking Expanded Movers against real mover locations; adding valid references to buffer
FOR ForCounterExit[GC.TRACK_SECTORS_STD][GC.OUTER_MERGE_COLLISION] := GC.nNumMinMovers TO GC.nNumMaxMovers DO
	IF AllRealSectorStatus[ForCounterExit[GC.TRACK_SECTORS_STD][GC.OUTER_MERGE_COLLISION]][GC.OUTER_MERGE_COLLISION].MoverIsOnSector THEN
			RealMoverIsOnSector[GC.OUTER_MERGE_COLLISION] := TRUE;
			EXIT;
		ELSIF NOT AllRealSectorStatus[ForCounterExit[GC.TRACK_SECTORS_STD][GC.OUTER_MERGE_COLLISION]][GC.OUTER_MERGE_COLLISION].MoverIsOnSector THEN
			RealMoverIsOnSector[GC.OUTER_MERGE_COLLISION] := FALSE;
		END_IF
END_FOR
END_METHOD

METHOD PRIVATE _M_VARINOUT_TroubleshootingJunk
VAR_INPUT
END_VAR
//IF ADR(TrackSectorsRef) <> 0 THEN
//	FOR MoverIndex := LowerOut TO UpperOut BY 1 DO

//AllSectorStatus[1][GC.OUTER_MERGE_COMBINED] 				:= TrackSectorsRef[1].SectorStatus[(GC.OUTER_MERGE_COMBINED)].MoverIsOnSector;
//AllSectorStatus[2][GC.OUTER_MERGE_COMBINED] 				:= TrackSectorsRef[2].SectorStatus[(GC.OUTER_MERGE_COMBINED)].MoverIsOnSector;
//AllSectorStatus[3][GC.OUTER_MERGE_COMBINED] 				:= TrackSectorsRef[3].SectorStatus[(GC.OUTER_MERGE_COMBINED)].MoverIsOnSector;
//AllSectorStatus[4][GC.OUTER_MERGE_COMBINED] 				:= TrackSectorsRef[4].SectorStatus[(GC.OUTER_MERGE_COMBINED)].MoverIsOnSector;
//AllSectorStatus[5][GC.OUTER_MERGE_COMBINED] 				:= TrackSectorsRef[5].SectorStatus[(GC.OUTER_MERGE_COMBINED)].MoverIsOnSector;
//AllSectorStatus[6][GC.OUTER_MERGE_COMBINED] 				:= TrackSectorsRef[6].SectorStatus[(GC.OUTER_MERGE_COMBINED)].MoverIsOnSector;
//AllSectorStatus[7][GC.OUTER_MERGE_COMBINED] 				:= TrackSectorsRef[7].SectorStatus[(GC.OUTER_MERGE_COMBINED)].MoverIsOnSector;
//AllSectorStatus[8][GC.OUTER_MERGE_COMBINED] 				:= TrackSectorsRef[8].SectorStatus[(GC.OUTER_MERGE_COMBINED)].MoverIsOnSector;
//AllSectorStatus[9][GC.OUTER_MERGE_COMBINED] 				:= TrackSectorsRef[9].SectorStatus[(GC.OUTER_MERGE_COMBINED)].MoverIsOnSector;
//AllSectorStatus[10][GC.OUTER_MERGE_COMBINED] 				:= TrackSectorsRef[10].SectorStatus[(GC.OUTER_MERGE_COMBINED)].MoverIsOnSector;
//AllSectorStatus[11][GC.OUTER_MERGE_COMBINED]				:= TrackSectorsRef[11].SectorStatus[(GC.OUTER_MERGE_COMBINED)].MoverIsOnSector;
//AllSectorStatus[12][GC.OUTER_MERGE_COMBINED]				:= TrackSectorsRef[12].SectorStatus[(GC.OUTER_MERGE_COMBINED)].MoverIsOnSector;
//AllSectorStatus[13][GC.OUTER_MERGE_COMBINED]				:= TrackSectorsRef[13].SectorStatus[(GC.OUTER_MERGE_COMBINED)].MoverIsOnSector;
//AllSectorStatus[14][GC.OUTER_MERGE_COMBINED]				:= TrackSectorsRef[14].SectorStatus[(GC.OUTER_MERGE_COMBINED)].MoverIsOnSector;
//AllSectorStatus[15][GC.OUTER_MERGE_COMBINED]				:= TrackSectorsRef[15].SectorStatus[(GC.OUTER_MERGE_COMBINED)].MoverIsOnSector;
//AllSectorStatus[16][GC.OUTER_MERGE_COMBINED] 				:= TrackSectorsRef[16].SectorStatus[(GC.OUTER_MERGE_COMBINED)].MoverIsOnSector;
//	END_FOR
//END_IF
END_METHOD

METHOD M_UpdateSectorCounts
VAR_INPUT
	SectorNr : UDINT; 
END_VAR
stSwitchStatus.ShuttleCountOnShortcut := 0;
IF ADR(TrackSectorsRef) <> 0 THEN // pointer validity check
	FOR ForCounterExit[GC.TRACK_SECTORS_STD][SectorNr] := GC.nNumMinMovers TO GVL_General.nNumMovers BY 1 DO

		stSwitchStatus.ShuttleCountOnShortcut		:= stSwitchStatus.ShuttleCountOnShortcut + TrackSectorsRef[ForCounterExit[GC.TRACK_SECTORS_STD][SectorNr]].SectorStatus[SectorNr].MoverCountOnSector;

	END_FOR
END_IF

//			IF TrackSectors[nForCounter].SectorStatus[GC.SHORTCUT_CALC_SECTOR_IPART].MoverEnteredSector.Q THEN
//				stSwitchStatus.ShuttleCountOnShortcut		:= stSwitchStatus.ShuttleCountOnShortcut + 1;
//			ELSIF TrackSectors[nForCounter].SectorStatus[GC.SHORTCUT_CALC_SECTOR_IPART].MoverExitedSector.Q THEN
//				stSwitchStatus.ShuttleCountOnShortcut		:= stSwitchStatus.ShuttleCountOnShortcut - 1;
//			END_IF
END_METHOD

PROPERTY P_AMoverIsOnSector : REFERENCE TO ARRAY[GC.MIN_SECTOR_CT..GC.MAX_SECTOR_CT] OF BOOL
GET
P_AMoverIsOnSector REF= RealMoverIsOnSector;
END_GET
END_PROPERTY

END_FUNCTION_BLOCK

// ---- POUs/FUNs/F_t_SL2a.TcPOU
FUNCTION F_t_SL2a : LREAL
VAR_INPUT
	SectorLength : LREAL;
	Acceleration : LREAL;
END_VAR
VAR
END_VAR

IF Acceleration <> 0 THEN
	F_t_SL2a := SQRT(SectorLength / (2*Acceleration));
END_IF

END_FUNCTION

// ---- POUs/FBs/FB_PlanarXtsMover.TcPOU
FUNCTION_BLOCK FB_PlanarXtsMover IMPLEMENTS RingBuffer.I_MoverBase, I_MoverSector (*, I_Mover *)

VAR_INPUT
	iTcIoXtsXpuMover			: REFERENCE TO Tc3_XTS_Utility.I_TcIoXtsXpuMover;
END_VAR

VAR
	stMoverOptions						: ST_MoverOptions;
	BaseMoveOptions						: Tc3_Mc3PlanarMotion.ST_MoveOnTrackOptions;
	GearInMasterMoverOptions	: Tc3_Mc3PlanarMotion.ST_GearInPosOnTrackWithMasterMoverOptions;
	
	MC_PlanarFeedbackGearInPosOnTrackWithMasterMover : Tc3_Mc3PlanarMotion.MC_PlanarFeedbackGearInPosOnTrackWithMasterMover;
		
	nMoverId			    				: UDINT;
	
	MoverFeedback							: Tc3_Mc3PlanarMotion.MC_PlanarFeedback;

	_McPlanarMover						: Tc3_Mc3PlanarMotion.MC_PlanarMover;
	_McPlanarTrackTrail    		: Tc3_Mc3PlanarMotion.MC_PlanarTrackTrail;
                        		
	stXtsPositionInfo					: Tc3_XTS_Utility.ST_PositionInfo;
	                      		
	Physics										: Tc3_Physics.PositionXYC;
	Dynamics									: Tc3_Physics.DynamicConstraint_PathXY;

	Mover				        			: MoverSort;
	
	IsUsingMagnet							: BOOL;
	
	SyncTrail 								: Tc3_Mc3PlanarMotion.MC_PlanarTrackTrail; 
	
	CmdDivert									: BOOL;
	eMerge										: E_MergeType;
	//InSync										: BOOL;
END_VAR

METHOD FB_init : BOOL
VAR_INPUT
	bInitRetains : BOOL; // if TRUE, the retain variables are initialized (warm start / cold start)
	bInCopyCode : BOOL;  // if TRUE, the instance afterwards gets moved into the copy code (online change)
END_VAR
stMoverOptions.BaseMoveOptions REF= BaseMoveOptions;
stMoverOptions.GearInMasterMoverOptions	REF= GearInMasterMoverOptions;

//Most options already initialized
//GearInMasterMoverOptions.allowedSlaveSyncDirections 				:= MC_SYNC_DIRECTIONS.Positive;
//GearInMasterMoverOptions.directionMasterSyncPosition				:= Tc3_Mc3PlanarMotion.MC_DIRECTION.mcDirectionNonModulo;
//GearInMasterMoverOptions.directionSlaveSyncPosition					:= Tc3_Mc3PlanarMotion.MC_DIRECTION.mcDirectionNonModulo;
//GearInMasterMoverOptions.followMover												:= FALSE;
GearInMasterMoverOptions.gap 																:= BaseMoveOptions.gap;
//GearInMasterMoverOptions.inSyncToleranceDistance						:= 0;
//GearInMasterMoverOptions.moduloToleranceMasterSyncPosition	:= 0;
//GearInMasterMoverOptions.moduloToleranceSlaveSyncPosition		:= 0;

syncTrail.AddTrack(track:= GVL_Mc3.MC_Tracks[E_TrackNum.Small]); 
syncTrail.AddTrack(track:= GVL_Mc3.MC_Tracks[E_TrackNum.Main]);
END_METHOD

METHOD Init : BOOL
VAR_INPUT

	XtsMover:   I_XtsXlMover1;
	XtsProcessingUnit :  I_XtsProcessingUnit1;
END_VAR



ipXtsMover:= XtsMover;
ipXtsProcessingUnit :=  XtsProcessingUnit;

stMoveOnTrackOptions.direction := MC_Direction.mcDirectionPositive;
stMoveOnTrackOptions.gapMode := MC_GAP_MODE_ON_TRACK.Fast1D;
stMoveOnTrackOptions.gap:= 800;

syncTrail.AddTrack(track:= GVL_Mc.MC_Tracks[E_TrackNum.Small]); 
syncTrail.AddTrack(track:= GVL_Mc.MC_Tracks[E_TrackNum.Main]); 


//_stDynamics.SetValuesVADJ(500, 4000, 4000, 10000);

bIsInitialized := TRUE;
END_METHOD

PROPERTY IsCommandedInShortcut : BOOL
GET
VAR
	nCounter: UDINT := 0;
END_VAR
_mcPlanarMover.GetTrackTrailInformation(_PlanarTrail);

IF _PlanarTrail.Error OR _PlanarTrail.Size < 1 THEN
   IsCommandedInShortcut := FALSE;
   RETURN;
END_IF
   
FOR nCounter := 0 TO _PlanarTrail.Size - 1 DO
	IF _PlanarTrail.GetTrackOidAt(nCounter) = GVL_Mc3.MC_Tracks[E_TrackNum.Small].MCTOPLC_STD.TrackOID  THEN
		IsCommandedInShortcut := TRUE;
		RETURN;
	END_IF
END_FOR

IsCommandedInShortcut := FALSE;
END_GET
END_PROPERTY

METHOD JoinTrack

VAR_INPUT
	feedback: REFERENCE TO MC_PlanarFeedback;
END_VAR

VAR_IN_OUT
	track: MC_PlanarTrack;
END_VAR
_McPlanarMover.JoinTrack(feedback, track, 0, 0);
END_METHOD

METHOD M_EvaluateGap
VAR_INPUT
	MoverIndex	: UDINT;
END_VAR
//IF TrackSectors[MoverIndex].SectorStatus[GC.OUTER_TIGHTGAP_ZONE].MoverIsOnSector OR
//TrackSectors[MoverIndex].SectorStatus[GC.INNER_MERGE_TO_FINISH].MoverIsOnSector THEN
//	fbPlanarXtsMover[MoverIndex].P_MoverOptions.BaseMoveOptions.gap := stMoverConfig.TightMoverGap;
//ELSIF TrackSectors[MoverIndex].SectorStatus[GC.OUTER_PRE_TG_ZONE].MoverIsOnSector THEN
//	fbPlanarXtsMover[MoverIndex].P_MoverOptions.TempGap := HelperFunctions.F_MapLReal(x := TrackSectors[MoverIndex].SectorStatus[GC.OUTER_PRE_TG_ZONE].PercentOfSectorTraversed,
//														in_min := 0.0, in_max := 1.0, out_min := stMoverConfig.NormalMoverGap, out_max := stMoverConfig.TightMoverGap);
//	fbPlanarXtsMover[MoverIndex].P_MoverOptions.BaseMoveOptions.gap := fbPlanarXtsMover[MoverIndex].P_MoverOptions.TempGap;
//ELSIF TrackSectors[MoverIndex].SectorStatus[GC.OUTER_POST_TG_ZONE].MoverIsOnSector THEN
//	fbPlanarXtsMover[MoverIndex].P_MoverOptions.TempGap := HelperFunctions.F_MapLReal(x := TrackSectors[MoverIndex].SectorStatus[GC.OUTER_POST_TG_ZONE].PercentOfSectorTraversed,
//														in_min := 0.0, in_max := 1.0, out_min := stMoverConfig.TightMoverGap, out_max := stMoverConfig.NormalMoverGap);
//	fbPlanarXtsMover[MoverIndex].P_MoverOptions.BaseMoveOptions.gap := fbPlanarXtsMover[MoverIndex].P_MoverOptions.TempGap;
//ELSE
	fbPlanarXtsMover[MoverIndex].P_MoverOptions.BaseMoveOptions.gap := stMoverConfig.NormalMoverGap;
//END_IF

IF fbPlanarXtsMover[MoverIndex].P_MoverOptions.BaseMoveOptions.gap = stMoverConfig.NormalMoverGap OR
	fbPlanarXtsMover[MoverIndex].P_MoverOptions.BaseMoveOptions.gap = stMoverConfig.TightMoverGap THEN
	fbPlanarXtsMover[MoverIndex].P_MoverOptions.GapInTransition := FALSE;
ELSE
	fbPlanarXtsMover[MoverIndex].P_MoverOptions.GapInTransition := TRUE;
END_IF
END_METHOD

PROPERTY P_CmdDivert : REFERENCE TO BOOL
GET
P_CmdDivert	REF= CmdDivert;
END_GET
END_PROPERTY

PROPERTY P_Dynamics : REFERENCE TO Tc3_Physics.DynamicConstraint_PathXY
GET
P_Dynamics	REF= Dynamics;
END_GET
END_PROPERTY

PROPERTY P_eMerge : REFERENCE TO E_MergeType
GET
P_eMerge	REF= eMerge;
END_GET
END_PROPERTY

PROPERTY P_InSync : REFERENCE TO BOOL
GET
P_InSync REF= MC_PlanarFeedbackGearInPosOnTrackWithMasterMover.inSync;
END_GET
END_PROPERTY

PROPERTY P_IsUsingMagnet : REFERENCE TO BOOL
GET
P_IsUsingMagnet REF= IsUsingMagnet;
END_GET
END_PROPERTY

PROPERTY P_MasterSyncId : REFERENCE TO UDINT
GET
P_MasterSyncId REF= stMoverOptions.MasterMoverID;
END_GET
END_PROPERTY

PROPERTY P_MasterSyncPosition : REFERENCE TO LREAL
GET
P_MasterSyncPosition REF= stMoverOptions.MasterSyncPosition;
END_GET
END_PROPERTY

PROPERTY P_MC_PlanarMover : REFERENCE TO Tc3_Mc3PlanarMotion.MC_PlanarMover
GET
P_MC_PlanarMover REF= _McPlanarMover;
END_GET
END_PROPERTY

PROPERTY P_MoverFeedback : REFERENCE TO Tc3_Mc3PlanarMotion.MC_PlanarFeedback
GET
P_MoverFeedback REF= MoverFeedback;
END_GET
END_PROPERTY

PROPERTY P_MoverId : UDINT
GET
P_MoverId	:= nMoverId;
END_GET
SET
nMoverId := P_MoverId;
END_SET
END_PROPERTY

PROPERTY P_MoverOptions : REFERENCE TO ST_MoverOptions
GET
P_MoverOptions REF= stMoverOptions;
END_GET
END_PROPERTY

PROPERTY P_MoverSort : REFERENCE TO MoverSort
GET
P_MoverSort	REF= Mover;
END_GET
END_PROPERTY

PROPERTY P_Physics : REFERENCE TO Tc3_Physics.PositionXYC
GET
P_Physics	REF= Physics;
END_GET
END_PROPERTY

PROPERTY P_PlanarFeedbackGearMM : REFERENCE TO Tc3_Mc3PlanarMotion.MC_PlanarFeedbackGearInPosOnTrackWithMasterMover
GET
P_PlanarFeedbackGearMM REF= MC_PlanarFeedbackGearInPosOnTrackWithMasterMover;
END_GET
END_PROPERTY

{warning 'Add property implementation'}
PROPERTY P_SectorsConfig : REFERENCE TO ST_SectorsConfig
GET
END_GET
END_PROPERTY

{warning 'Add property implementation'}
PROPERTY P_SectorsStatus : REFERENCE TO ST_SectorsStatus
GET
END_GET
END_PROPERTY

PROPERTY P_SyncTrail : REFERENCE TO Tc3_Mc3PlanarMotion.MC_PlanarTrackTrail
GET
P_SyncTrail REF= SyncTrail;
END_GET
END_PROPERTY

PROPERTY P_TrackConfig : REFERENCE TO ST_TrackConfig
GET
END_GET
END_PROPERTY

PROPERTY P_XtsPositionInfo : REFERENCE TO Tc3_XTS_Utility.ST_PositionInfo
GET
P_XtsPositionInfo	REF= stXtsPositionInfo;
END_GET
END_PROPERTY

METHOD SyncToOtherMover : BOOL
VAR_INPUT
	masterSyncPos : LREAL; // Position on the master track
	followerSyncPos : LREAL; // position on the follower track
	PlanarMoverToFollow: REFERENCE TO Tc3_Mc3PlanarMotion.MC_PlanarMover;
	masterTrack : REFERENCE TO Tc3_Mc3PlanarMotion.MC_PlanarTrack; 
	followerTrack : REFERENCE TO Tc3_Mc3PlanarMotion.MC_PlanarTrack; 
	velo : LREAL; 
END_VAR

VAR
	trail: Tc3_Mc3PlanarMotion.MC_PlanarTrackTrail;

END_VAR
//Options.allowedSlaveSyncDirections := MC_SYNC_DIRECTIONS.Positive; 
//options.directionMasterSyncPosition := MC_DIRECTION.mcDirectionNonModulo; 
//options.directionSlaveSyncPosition := MC_DIRECTION.mcDirectionNonModulo;  
//options.followMover := FALSE; 
//options.gap := 0; // elimnate gap funciton 
//options.inSyncToleranceDistance :=0; 
//options.moduloToleranceMasterSyncPosition := 0; 
//options.moduloToleranceSlaveSyncPosition := 0;  
//_stDynamics.V := velo; 

fbPlanarMover.GearInPosOnTrackWithMasterMover(
//	commandFeedback:=  SyncMoverFeedback , 
//	masterMover:= PlanarMoverToFollow , 
//	trackTrail:= syncTrail, // may need to give a trail maybe not
//	masterSyncPosition:= masterSyncPos, 
//	masterSyncPositionTrack:= MasterTrack , 
//	slaveSyncPosition:= followerSyncPos, 
//	slaveSyncPositionTrack:= followerTrack, 
//	constraint:=_stDynamics , 
//	options:=options );
END_METHOD

METHOD Update : PVOID
IF iTcIoXtsXpuMover <> 0 THEN
  stXtsPositionInfo	:= iTcIoXtsXpuMover.GetPositionInfo();
END_IF

_mcPlanarMover.Update();

IF eMerge = E_MergeType.FlyingMergeMoveSyncd OR eMerge = E_MergeType.MergeFromStaticSyncd THEN
	MC_PlanarFeedbackGearInPosOnTrackWithMasterMover.Update();
END_IF

_mcPlanarMover.GetTrackTrailInformation(_McPlanarTrackTrail);

Mover.MoverNumber 	:= nMoverId;
Mover.MoverPos    	:= _McPlanarMover.MCTOPLC.SETONTRACK.SetPos;
Mover.TrackID     	:= _McPlanarMover.MCTOPLC.SETONTRACK.TrackOID;
//MoverPhysics		:= 

{warning <'Method Not Called'>}
//_M_UpdateStatus();

IF _McPlanarTrackTrail.Error OR _McPlanarTrackTrail.Size <= 1 THEN
   RETURN;
END_IF

IF iTcIoXtsXpuMover <> 0 THEN
  //SmallCircle
  IF _McPlanarTrackTrail.GetTrackOidAt(1) = MC_Tracks[E_TrackNum.Small].MCTOPLC_STD.TrackOID   THEN
    iTcIoXtsXpuMover.SetActiveTrackObjectId(XtsCompleteTrackInnerOID);
  //BigCircle
  ELSIF _McPlanarTrackTrail.GetTrackOidAt(1) =MC_Tracks[E_TrackNum.Big].MCTOPLC_STD.TrackOID THEN
    iTcIoXtsXpuMover.SetActiveTrackObjectId(XtsCompleteTrackOuterOID);
  END_IF
END_IF
END_METHOD

END_FUNCTION_BLOCK

// ---- POUs/FBs/FB_ExpandedMover.TcPOU
FUNCTION_BLOCK FB_ExpandedMover
VAR_INPUT
	MoverRef		: REFERENCE TO FB_PlanarXtsMover;
END_VAR
VAR
	eExpMoverConfig		: RingBuffer.E_ExpMover;
	stExpMoverStatus		: ST_ExpMoverStatus;
END_VAR

_M_UpdatePositions();

METHOD PROTECTED _M_UpdatePositions
IF ADR(MoverRef) <> 0 THEN
	stExpMoverStatus.XtsBaseRefData 							 REF= MoverRef.P_XtsPositionInfo;
	stExpMoverStatus.XtsAdjustedData.nPartObjectid	:= stExpMoverStatus.XtsBaseRefData.nPartObjectid;
	stExpMoverStatus.XtsAdjustedData.nTrackObjectid	:= stExpMoverStatus.XtsBaseRefData.nTrackObjectid;
	IF eExpMoverConfig = RingBuffer.E_ExpMover.Head THEN
		stExpMoverStatus.TrackSectorBndryHeadF 		:= stExpMoverStatus.XtsBaseRefData.fTrackPosition + stTrackGlobalConfig.ExpMoverLength + GC.SHUTTLE_LENGTH/2;
		stExpMoverStatus.TrackSectorCenterHead 		:= stExpMoverStatus.XtsBaseRefData.fTrackPosition + stTrackGlobalConfig.ExpMoverLength + GC.SHUTTLE_LENGTH/2;
		stExpMoverStatus.XtsAdjustedData.fTrackPosition	:= stExpMoverStatus.TrackSectorCenterHead;
		stExpMoverStatus.TrackSectorBndryHeadR 		:= stExpMoverStatus.XtsBaseRefData.fTrackPosition + GC.SHUTTLE_LENGTH/2;
		stExpMoverStatus.PartSectorBndryHeadF 		:= stExpMoverStatus.XtsBaseRefData.fPartPosition + stTrackGlobalConfig.ExpMoverLength + GC.SHUTTLE_LENGTH/2;
		stExpMoverStatus.PartSectorCenterHead 		:= stExpMoverStatus.XtsBaseRefData.fPartPosition + stTrackGlobalConfig.ExpMoverLength + GC.SHUTTLE_LENGTH/2;
		stExpMoverStatus.XtsAdjustedData.fPartPosition	:= stExpMoverStatus.PartSectorCenterHead;
		stExpMoverStatus.PartSectorBndryHeadR 		:= stExpMoverStatus.XtsBaseRefData.fPartPosition + GC.SHUTTLE_LENGTH/2;
	ELSIF eExpMoverConfig = RingBuffer.E_ExpMover.Tail THEN
		stExpMoverStatus.TrackSectorBndryTailF		:= stExpMoverStatus.XtsBaseRefData.fTrackPosition - GC.SHUTTLE_LENGTH/2;
		stExpMoverStatus.TrackSectorCenterTail		:= stExpMoverStatus.XtsBaseRefData.fTrackPosition - stTrackGlobalConfig.ExpMoverLength - GC.SHUTTLE_LENGTH/2;
		stExpMoverStatus.XtsAdjustedData.fTrackPosition	:= stExpMoverStatus.TrackSectorCenterTail;
		stExpMoverStatus.TrackSectorBndryTailR		:= stExpMoverStatus.XtsBaseRefData.fTrackPosition - stTrackGlobalConfig.ExpMoverLength - GC.SHUTTLE_LENGTH/2;
		stExpMoverStatus.PartSectorBndryTailF			:= stExpMoverStatus.XtsBaseRefData.fPartPosition - GC.SHUTTLE_LENGTH/2;
		stExpMoverStatus.PartSectorCenterTail			:= stExpMoverStatus.XtsBaseRefData.fPartPosition - stTrackGlobalConfig.ExpMoverLength - GC.SHUTTLE_LENGTH/2;
		stExpMoverStatus.XtsAdjustedData.fPartPosition	:= stExpMoverStatus.PartSectorCenterTail;
		stExpMoverStatus.PartSectorBndryTailR			:= stExpMoverStatus.XtsBaseRefData.fPartPosition - stTrackGlobalConfig.ExpMoverLength - GC.SHUTTLE_LENGTH/2;
	END_IF
END_IF
END_METHOD

PROPERTY P_ExpMoverConfig : REFERENCE TO RingBuffer.E_ExpMover
GET
P_ExpMoverConfig REF= eExpMoverConfig;
END_GET
END_PROPERTY

PROPERTY P_ExpMoverStatus : REFERENCE TO ST_ExpMoverStatus
GET
P_ExpMoverStatus REF= stExpMoverStatus;
END_GET
END_PROPERTY

END_FUNCTION_BLOCK

// ---- POUs/FBs/FB_AllExpMovers.TcPOU
FUNCTION_BLOCK FB_AllExpMovers
VAR_INPUT
	HeadMoversRef					: REFERENCE TO ARRAY[GC.nNumMinMovers..GC.nNumMaxMovers] OF FB_ExpandedMover;
	TailMoversRef					: REFERENCE TO ARRAY[GC.nNumMinMovers..GC.nNumMaxMovers] OF FB_ExpandedMover;
END_VAR
VAR
	MoverIndex					: UDINT;
	ForCounterExit 			: ARRAY[GC.MIN_SECTOR_CT..GC.MAX_SECTOR_CT] OF UDINT;
	SectorIndex 				: UDINT;
//	LapTrig1						: ST_MergeWindow;
//	LapGap							: ST_MergeWindow;
//	WindowClearDebounce : TIME;
//	GapClearTail				: Tc2_Standard.TON;

//	AMoverIsOnVoid			:	ARRAY[GC.MIN_SECTOR_CT..GC.MAX_SECTOR_CT] OF BOOL;
END_VAR
VAR CONSTANT
	CONVERT_MS_100NS_COUNT	: LREAL := 1E4;
END_VAR

_M_Configuration();

//_M_EvaluateStatus();

METHOD PRIVATE _M_Configuration
FOR MoverIndex := GC.nNumMinMovers TO GC.nNumMaxMovers DO
	HeadMoversRef[MoverIndex].P_ExpMoverConfig := RingBuffer.E_ExpMover.Head;
	TailMoversRef[MoverIndex].P_ExpMoverConfig := RingBuffer.E_ExpMover.Tail;
END_FOR
END_METHOD

METHOD PRIVATE _M_EvaluateStatus
END_METHOD

METHOD PRIVATE _M_EvaluateStatus1
IF ADR(TrackSectorsRef) <> 0 THEN // pointer validity check
	FOR MoverIndex := GC.nNumMinMovers TO GVL_General.nNumMovers BY 1 DO
		FOR SectorIndex := GC.MIN_SECTOR_CT TO GC.MAX_SECTOR_CT BY 1 DO
			
//			IF LapTrig1.Latch AND_THEN TrackSectorsRef[MoverIndex].SectorStatus[GC.OUTER_FINISH_MOVERTOFOLLOW].MoverIsOnSector THEN
//				MoverIdToFollowOnMerge	:= MoverIndex;
//			END_IF
	
		END_FOR
	END_FOR
END_IF

//Merge Combined
//FOR ForCounterExit[GC.OUTER_MERGE_INFRONT] := GC.nNumMinMovers TO GVL_General.nNumMovers BY 1 DO
//	IF AllSectorStatus[ForCounterExit[GC.OUTER_MERGE_INFRONT]][GC.OUTER_MERGE_INFRONT].MoverIsOnSector THEN
//			AMoverIsOnSector[GC.OUTER_MERGE_INFRONT] := TRUE;
//			EXIT;
//		ELSIF NOT AllSectorStatus[ForCounterExit[GC.OUTER_MERGE_INFRONT]][GC.OUTER_MERGE_INFRONT].MoverIsOnSector THEN
//			AMoverIsOnSector[GC.OUTER_MERGE_INFRONT] := FALSE;
//		END_IF
//END_FOR

//Lap Trig 1
FOR ForCounterExit[GC.OUTER_FINISH_LAPTRIG] := GC.nNumMinMovers TO GVL_General.nNumMovers BY 1 DO
//		IF AllSectorStatus[ForCounterExit[GC.OUTER_FINISH_LAPTRIG1]][GC.OUTER_FINISH_LAPTRIG1].MoverIsOnSector THEN
//			AMoverIsOnSector[GC.OUTER_FINISH_LAPTRIG1] := TRUE;
//			EXIT;
//		ELSIF NOT AllSectorStatus[ForCounterExit[GC.OUTER_FINISH_LAPTRIG1]][GC.OUTER_FINISH_LAPTRIG1].MoverIsOnSector THEN
//			AMoverIsOnSector[GC.OUTER_FINISH_LAPTRIG1] := FALSE;
//		END_IF
	IF NOT LapTrig1.Latch AND NOT LapGap.Latch AND AllSectorStatus[ForCounterExit[GC.OUTER_FINISH_LAPTRIG]][GC.OUTER_FINISH_LAPTRIG].MoverExitedSector.Q THEN
			LapTrig1.Latch := TRUE;
			GapClearTail.IN	:= TRUE;
			LapTrig1.timestamp	:= Tc2_System.F_GetSystemTime();
			EXIT;
		END_IF
	IF LapTrig1.Latch AND NOT LapGap.Latch AND AllSectorStatus[ForCounterExit[GC.OUTER_FINISH_LAPTRIG]][GC.OUTER_FINISH_LAPTRIG].MoverEnteredSector.Q THEN
			LapGap.Latch := TRUE;
			LapGap.timestamp	:= Tc2_System.F_GetSystemTime();
			EXIT;
		END_IF
		
END_FOR

//Lap Trig 2
//FOR ForCounterExit[GC.OUTER_FINISH_LAPTRIG2] := GC.nNumMinMovers TO GVL_General.nNumMovers BY 1 DO
//		IF AllSectorStatus[ForCounterExit[GC.OUTER_FINISH_LAPTRIG2]][GC.OUTER_FINISH_LAPTRIG2].MoverIsOnSector THEN
//			AMoverIsOnSector[GC.OUTER_FINISH_LAPTRIG2] := TRUE;
//			EXIT;
//		ELSIF NOT AllSectorStatus[ForCounterExit[GC.OUTER_FINISH_LAPTRIG2]][GC.OUTER_FINISH_LAPTRIG2].MoverIsOnSector THEN
//			AMoverIsOnSector[GC.OUTER_FINISH_LAPTRIG2] := FALSE;
//		END_IF
//	IF LapTrig1.Latch AND NOT LapTrig2.Latch AND_THEN AllSectorStatus[ForCounterExit[GC.OUTER_FINISH_LAPTRIG2]][GC.OUTER_FINISH_LAPTRIG2].MoverEnteredSector.Q THEN
//			LapTrig2.Latch := TRUE;
//			EXIT;
//		END_IF
//END_FOR

_M_EvaluateWindow();

GapClearTail(PT := WindowClearDebounce);
END_METHOD

METHOD PRIVATE _M_EvaluateWindow
VAR_INST
	TrigAdd : BOOL;
	TrigRem : BOOL;
	DistanceDeltaFromMerge : LREAL;
	TempCalc : LREAL;
END_VAR
IF (stMoverConfig.NormalVelo - stMoverConfig.VeloComp) <> 0 THEN
	WindowClearDebounce := LREAL_TO_TIME(1000*stTrackGlobalConfig.ExpMoverLength / (stMoverConfig.NormalVelo - stMoverConfig.VeloComp));
END_IF

IF LapTrig1.Latch AND LapGap.Latch THEN
//	TimeDeltaTemp	:= LapGap.timestamp - LapTrig1.timestamp;
//	TimeDelta := ULINT_TO_REAL(TimeDeltaTemp) / TicksPerS;

	LapTrig1.Latch := FALSE;
	LapGap.Latch := FALSE;
	GapClearTail.IN	:= FALSE;

END_IF

IF GapClearTail.Q AND NOT LapGap.Latch THEN
	// Position to match with merging mover
	LapTrig1.timestamp;
//	MergeQueue.AddObjToBuffer(RefObject := );
	GapClearTail.IN	:= FALSE;
END_IF

//DistanceDeltaFromMerge := GVL_Mc3.MC_Tracks[E_TrackNum.Big].GetLength() - ValidPosnTime.ValidPosnSrc;
IF (stMoverConfig.NormalVelo - stMoverConfig.VeloComp) <> 0 THEN 
	TempCalc 	:= 1000* (DistanceDeltaFromMerge / (stMoverConfig.NormalVelo - stMoverConfig.VeloComp));
END_IF
//TargetTimeForLastTPosnAtMerge	:= MergeQueue.P_LastObjectRemoved + LREAL_TO_ULINT(TempCalc * CONVERT_MS_100NS_COUNT);  //ms to count of 100ns intervals

//ValidPosnTime.ValidTargetDestTime := MergeQueue.P_LastObjectRemoved + ;

IF TrigRem THEN
	TrigRem	:= FALSE;
	MergeQueue.RemoveObjFromBuffer();
END_IF

IF TrigAdd THEN
	TrigAdd	:= FALSE;
	MergeQueue.AddObjToBuffer(RefObject := ValidMergeObject);	
END_IF

//Make a dynamic sector that follows the "virtual" position; could be used as a PermIntlk for violation of the sector by a real mover;
END_METHOD

END_FUNCTION_BLOCK

// ---- POUs/FBs/FB_MoverLists.TcPOU
FUNCTION_BLOCK FB_MoverLists
VAR_INPUT
END_VAR
VAR_OUTPUT
END_VAR
VAR
	aitfMovers : ARRAY[GC.nNumMinMovers..GVL_General.nNumMovers] OF I_Mover;
	SectorIndex	: UDINT;
	MoverIndex	: UDINT;
END_VAR

FOR SectorIndex := GC.MIN_SECTOR_CT TO gc.MAX_SECTOR_CT BY 1 DO
	FOR MoverIndex := GC.nNumMinMovers TO GVL_General.nNumMovers BY 1 DO
		aitfMovers[GC.nNumMinMovers].P_TrackSectors.SectorStatus[SectorIndex].PercentOfSectorTraversed;
	END_FOR
END_FOR

//

END_FUNCTION_BLOCK

// ---- POUs/FBs/FB_MoveState.TcPOU
FUNCTION_BLOCK FB_MoveState
VAR_INPUT
	fbPlanarXtsMover 	: REFERENCE TO FB_PlanarXtsMover;
	TrackSectors			: REFERENCE TO FB_TrackSectors;
END_VAR
VAR_OUTPUT
END_VAR
//Make Stateless
VAR
	nMoveState	: UDINT;
END_VAR

//Make Stateless
M_EvaluateTrackTransition(DepartingTrackRef := E_TrackNum.Main, ArrivingTrackRef := E_TrackNum.Big, DepartPermissiveSectorRef := );

M_EvaluateTrackTransition(DepartingTrackRef := E_TrackNum.Big, ArrivingTrackRef := E_TrackNum.Main, DepartPermissiveSectorRef := );

M_EvaluateTrackTransition(DepartingTrackRef := E_TrackNum.Main, ArrivingTrackRef := E_TrackNum.Small, DepartPermissiveSectorRef := );

M_EvaluateTrackTransition(DepartingTrackRef := E_TrackNum.Small, ArrivingTrackRef := E_TrackNum.Main, DepartPermissiveSectorRef := );


CASE nMoveState OF
				
